# B&R Automation Studio project 2SegDemo
Automation Studio 4.10.2.37; technology packages: mapp 5.14.1, mappCockpit 5.14.0, mappControl 5.14.1, mappMotion 5.14.2, mappView 5.14.2

## Configuration 1685

CPU X20CP1685, AutomationRuntime C4.90, Build 6.3.0, Safety 1.10, Vc V4.72.2

### Task classes (Cpu.sw)
```
Cyclic#1 (cycle 1000 us, tolerance 0 us):
  6DCtrl <- Source.6DCtrl.6DCtrl.prg
  VarDemos <- Source.Demos.VarDemos.prg
  AntiSlosh <- Source.Demos.AntiSlosh.prg
Cyclic#3:
  Main <- Source.Main.Main.prg
Cyclic#4:
  Recovery <- Source.ShuttleCtrl.Recovery.prg
Cyclic#8 (cycle 1000 us):
  Vis <- Source.Auxil.Vis.prg
  MacroLoad <- Source.6DCtrl.MacroLoad.prg
  Monitor6D <- Source.Auxil.Monitor6D.prg
DataObjects: McAcpSys
Binaries: mvLoader, McMechSys, McProfGen, TCData, McAcpSim, mCoWebSc, FWRules, McAcpDrv, udbdef, TCLang, arcoal, arflatprv, arsvcreg, OpcUaSrv, Role, arconfig, Settings, User, asfw, ashwd, Config_1, ashwac, sysconf, Config, Config_2, iomap, TC, TraceConfi, Config_3, Config_4, Hierarchy
Libraries: runtime, brsystem, sys_lib, CoTrace, FileIO, AsZip, McPureVAx, operator, astime, AsIecCon, standard, McAcp6D, AsMath, AsXml, AsBrStr, AsIODiag, LoggingLib, asstring, ArEventLog, AsTCP, snprintf, MTTypes, AsBrMath, McBase, McAcpAx, McAxis, MpAxis, MpBase, MpAudit, MpRecipe, MpFile, MTFilter, MTBasics, MpServer, MpAlarmX, SlFreeBase, MTProfile, asepl, aruser, dataobj, powerlnk, arssl, asusb, WFilter, asarlog, asmem, asarprof, asio, McPathGen, McProgInt, McAxGroup, MpRobotics, McAcpTrak
```

### Hardware
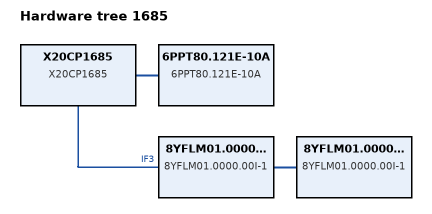
```
6PPT80.121E-10A : 6PPT80.121E-10A v1.0.2.0  [ETH1 -> X20CP1685.IF2 [Cable Type=PowerlinkCable, Length=10, Version=1.0.0.3]]
  Terminal = true
  Mode = Manual
  InternetAddress = 192.168.10.85
  Subnetmask = 255.255.255.0
  PasswordVNC = 
  PasswordCIFS = 
  PasswordService = 
8YFLM01.0000.00I-1 : 8YFLM01.0000.00I-1 v0.0.0.1  [PLK1 -> X20CP1685.IF3 (NodeNumber=101) [Cable Type=PowerlinkCable, Length=10, Version=1.0.0.3]; PLK2 -> 8YFLM01.0000.00I-1a.PLK1 (NodeNumber=101) [Cable Type=PowerlinkCable, Length=10, Version=1.0.0.3]]
  Supervision = off
8YFLM01.0000.00I-1a : 8YFLM01.0000.00I-1 v0.0.0.1 (Disabled=true)  [PLK1 -> 8YFLM01.0000.00I-1.PLK2 (NodeNumber=102) [Cable Type=PowerlinkCable, Length=10, Version=1.0.0.3]]
  Supervision = off
X20CP1685 : X20CP1685 v1.4.0.0
  Connector IF2:
    ActivateDevice = 1
    Mode = Manual
    InternetAddress = 192.168.10.82
    SubnetMask = 255.255.255.0
    ActivateSnmp = 2
  Connector IF3:
    CycleTime = 1000
  Connector IF6:
    ActivateX2X = 0
  ConfigurationID = OnsiteDemo_1685
  UserPartitionSize = 10
  TimerDeviceType = EPLX2X
  TimerDevice = X20CP1685.IF3
  Cyclic1Duration = 1000
  Cyclic1Tolerance = 0
  Cyclic1Stack = 75536
  Cyclic1Output = 1
  Cyclic2Duration = 10000
  Cyclic2Tolerance = 10000
  Cyclic8Duration = 1000
  FileDevice1
  FileDeviceName1 = CNC_PrgDir
  FileDevicePath1 = F:/Programs
  FileDevice2
  FileDeviceName2 = 6DMacro
  FileDevicePath2 = F:/Macros
  FtpUser1
  FtpUsername1 = user
  FtpUserPassword1 = OnC+KhD/SpTljM37peNi/Txa+vmo0PgBkRCvsZXBTJk=  // user
  FtpUserSalt1 = 0mgKB/Te
  FTPAccessRight1 = 0
  ActivateOpcUa = 1
  OpcUaPort = 4841
  OpcUaInformationModels_PV_Version = 2
```

### IoMap.iom - X20CP1685/IoMap.iom
```iecst
VAR_CONFIG
	Cyclic#1.::FBin[0] AT %IW."8YFLM01.0000.00I-1".EPL_FB_IN_0_I2007_S01;
	Cyclic#1.::FBin[1] AT %IW."8YFLM01.0000.00I-1".EPL_FB_IN_1_I2007_S02;
	Cyclic#1.::FBin[10] AT %IW."8YFLM01.0000.00I-1".EPL_FB_IN_10_I2007_S0B;
	Cyclic#1.::FBin[100] AT %IW."8YFLM01.0000.00I-1".EPL_FB_IN_100_I2007_S65;
	Cyclic#1.::FBin[101] AT %IW."8YFLM01.0000.00I-1".EPL_FB_IN_101_I2007_S66;
	Cyclic#1.::FBin[102] AT %IW."8YFLM01.0000.00I-1".EPL_FB_IN_102_I2007_S67;
	Cyclic#1.::FBin[103] AT %IW."8YFLM01.0000.00I-1".EPL_FB_IN_103_I2007_S68;
	Cyclic#1.::FBin[104] AT %IW."8YFLM01.0000.00I-1".EPL_FB_IN_104_I2007_S69;
	Cyclic#1.::FBin[105] AT %IW."8YFLM01.0000.00I-1".EPL_FB_IN_105_I2007_S6A;
	Cyclic#1.::FBin[106] AT %IW."8YFLM01.0000.00I-1".EPL_FB_IN_106_I2007_S6B;
	Cyclic#1.::FBin[107] AT %IW."8YFLM01.0000.00I-1".EPL_FB_IN_107_I2007_S6C;
	Cyclic#1.::FBin[108] AT %IW."8YFLM01.0000.00I-1".EPL_FB_IN_108_I2007_S6D;
	Cyclic#1.::FBin[109] AT %IW."8YFLM01.0000.00I-1".EPL_FB_IN_109_I2007_S6E;
	Cyclic#1.::FBin[11] AT %IW."8YFLM01.0000.00I-1".EPL_FB_IN_11_I2007_S0C;
	Cyclic#1.::FBin[110] AT %IW."8YFLM01.0000.00I-1".EPL_FB_IN_110_I2007_S6F;
	Cyclic#1.::FBin[111] AT %IW."8YFLM01.0000.00I-1".EPL_FB_IN_111_I2007_S70;
	Cyclic#1.::FBin[112] AT %IW."8YFLM01.0000.00I-1".EPL_FB_IN_112_I2007_S71;
	Cyclic#1.::FBin[113] AT %IW."8YFLM01.0000.00I-1".EPL_FB_IN_113_I2007_S72;
	Cyclic#1.::FBin[114] AT %IW."8YFLM01.0000.00I-1".EPL_FB_IN_114_I2007_S73;
	Cyclic#1.::FBin[115] AT %IW."8YFLM01.0000.00I-1".EPL_FB_IN_115_I2007_S74;
	Cyclic#1.::FBin[116] AT %IW."8YFLM01.0000.00I-1".EPL_FB_IN_116_I2007_S75;
	Cyclic#1.::FBin[117] AT %IW."8YFLM01.0000.00I-1".EPL_FB_IN_117_I2007_S76;
	Cyclic#1.::FBin[118] AT %IW."8YFLM01.0000.00I-1".EPL_FB_IN_118_I2007_S77;
	Cyclic#1.::FBin[119] AT %IW."8YFLM01.0000.00I-1".EPL_FB_IN_119_I2007_S78;
	Cyclic#1.::FBin[12] AT %IW."8YFLM01.0000.00I-1".EPL_FB_IN_12_I2007_S0D;
	Cyclic#1.::FBin[120] AT %IW."8YFLM01.0000.00I-1".EPL_FB_IN_120_I2007_S79;
	Cyclic#1.::FBin[121] AT %IW."8YFLM01.0000.00I-1".EPL_FB_IN_121_I2007_S7A;
	Cyclic#1.::FBin[122] AT %IW."8YFLM01.0000.00I-1".EPL_FB_IN_122_I2007_S7B;
	Cyclic#1.::FBin[123] AT %IW."8YFLM01.0000.00I-1".EPL_FB_IN_123_I2007_S7C;
	Cyclic#1.::FBin[124] AT %IW."8YFLM01.0000.00I-1".EPL_FB_IN_124_I2007_S7D;
	Cyclic#1.::FBin[125] AT %IW."8YFLM01.0000.00I-1".EPL_FB_IN_125_I2007_S7E;
	Cyclic#1.::FBin[126] AT %IW."8YFLM01.0000.00I-1".EPL_FB_IN_126_I2007_S7F;
	Cyclic#1.::FBin[127] AT %IW."8YFLM01.0000.00I-1".EPL_FB_IN_127_I2007_S80;
	Cyclic#1.::FBin[128] AT %IW."8YFLM01.0000.00I-1".EPL_FB_IN_128_I2007_S81;
	Cyclic#1.::FBin[129] AT %IW."8YFLM01.0000.00I-1".EPL_FB_IN_129_I2007_S82;
	Cyclic#1.::FBin[13] AT %IW."8YFLM01.0000.00I-1".EPL_FB_IN_13_I2007_S0E;
	Cyclic#1.::FBin[130] AT %IW."8YFLM01.0000.00I-1".EPL_FB_IN_130_I2007_S83;
	Cyclic#1.::FBin[131] AT %IW."8YFLM01.0000.00I-1".EPL_FB_IN_131_I2007_S84;
	Cyclic#1.::FBin[132] AT %IW."8YFLM01.0000.00I-1".EPL_FB_IN_132_I2007_S85;
	Cyclic#1.::FBin[133] AT %IW."8YFLM01.0000.00I-1".EPL_FB_IN_133_I2007_S86;
	Cyclic#1.::FBin[134] AT %IW."8YFLM01.0000.00I-1".EPL_FB_IN_134_I2007_S87;
	Cyclic#1.::FBin[135] AT %IW."8YFLM01.0000.00I-1".EPL_FB_IN_135_I2007_S88;
	Cyclic#1.::FBin[136] AT %IW."8YFLM01.0000.00I-1".EPL_FB_IN_136_I2007_S89;
	Cyclic#1.::FBin[137] AT %IW."8YFLM01.0000.00I-1".EPL_FB_IN_137_I2007_S8A;
	Cyclic#1.::FBin[138] AT %IW."8YFLM01.0000.00I-1".EPL_FB_IN_138_I2007_S8B;
	Cyclic#1.::FBin[139] AT %IW."8YFLM01.0000.00I-1".EPL_FB_IN_139_I2007_S8C;
	Cyclic#1.::FBin[14] AT %IW."8YFLM01.0000.00I-1".EPL_FB_IN_14_I2007_S0F;
	Cyclic#1.::FBin[140] AT %IW."8YFLM01.0000.00I-1".EPL_FB_IN_140_I2007_S8D;
	Cyclic#1.::FBin[141] AT %IW."8YFLM01.0000.00I-1".EPL_FB_IN_141_I2007_S8E;
	Cyclic#1.::FBin[142] AT %IW."8YFLM01.0000.00I-1".EPL_FB_IN_142_I2007_S8F;
	Cyclic#1.::FBin[143] AT %IW."8YFLM01.0000.00I-1".EPL_FB_IN_143_I2007_S90;
	Cyclic#1.::FBin[144] AT %IW."8YFLM01.0000.00I-1".EPL_FB_IN_144_I2007_S91;
	Cyclic#1.::FBin[145] AT %IW."8YFLM01.0000.00I-1".EPL_FB_IN_145_I2007_S92;
	Cyclic#1.::FBin[146] AT %IW."8YFLM01.0000.00I-1".EPL_FB_IN_146_I2007_S93;
	Cyclic#1.::FBin[147] AT %IW."8YFLM01.0000.00I-1".EPL_FB_IN_147_I2007_S94;
	Cyclic#1.::FBin[148] AT %IW."8YFLM01.0000.00I-1".EPL_FB_IN_148_I2007_S95;
	Cyclic#1.::FBin[149] AT %IW."8YFLM01.0000.00I-1".EPL_FB_IN_149_I2007_S96;
	Cyclic#1.::FBin[15] AT %IW."8YFLM01.0000.00I-1".EPL_FB_IN_15_I2007_S10;
	Cyclic#1.::FBin[150] AT %IW."8YFLM01.0000.00I-1".EPL_FB_IN_150_I2007_S97;
	Cyclic#1.::FBin[151] AT %IW."8YFLM01.0000.00I-1".EPL_FB_IN_151_I2007_S98;
	Cyclic#1.::FBin[152] AT %IW."8YFLM01.0000.00I-1".EPL_FB_IN_152_I2007_S99;
	Cyclic#1.::FBin[153] AT %IW."8YFLM01.0000.00I-1".EPL_FB_IN_153_I2007_S9A;
	Cyclic#1.::FBin[154] AT %IW."8YFLM01.0000.00I-1".EPL_FB_IN_154_I2007_S9B;
	Cyclic#1.::FBin[155] AT %IW."8YFLM01.0000.00I-1".EPL_FB_IN_155_I2007_S9C;
	Cyclic#1.::FBin[156] AT %IW."8YFLM01.0000.00I-1".EPL_FB_IN_156_I2007_S9D;
	Cyclic#1.::FBin[157] AT %IW."8YFLM01.0000.00I-1".EPL_FB_IN_157_I2007_S9E;
	Cyclic#1.::FBin[158] AT %IW."8YFLM01.0000.00I-1".EPL_FB_IN_158_I2007_S9F;
	Cyclic#1.::FBin[159] AT %IW."8YFLM01.0000.00I-1".EPL_FB_IN_159_I2007_SA0;
	Cyclic#1.::FBin[16] AT %IW."8YFLM01.0000.00I-1".EPL_FB_IN_16_I2007_S11;
	Cyclic#1.::FBin[160] AT %IW."8YFLM01.0000.00I-1".EPL_FB_IN_160_I2007_SA1;
	Cyclic#1.::FBin[161] AT %IW."8YFLM01.0000.00I-1".EPL_FB_IN_161_I2007_SA2;
	Cyclic#1.::FBin[162] AT %IW."8YFLM01.0000.00I-1".EPL_FB_IN_162_I2007_SA3;
	Cyclic#1.::FBin[163] AT %IW."8YFLM01.0000.00I-1".EPL_FB_IN_163_I2007_SA4;
	Cyclic#1.::FBin[164] AT %IW."8YFLM01.0000.00I-1".EPL_FB_IN_164_I2007_SA5;
	Cyclic#1.::FBin[165] AT %IW."8YFLM01.0000.00I-1".EPL_FB_IN_165_I2007_SA6;
	Cyclic#1.::FBin[166] AT %IW."8YFLM01.0000.00I-1".EPL_FB_IN_166_I2007_SA7;
	Cyclic#1.::FBin[167] AT %IW."8YFLM01.0000.00I-1".EPL_FB_IN_167_I2007_SA8;
	Cyclic#1.::FBin[168] AT %IW."8YFLM01.0000.00I-1".EPL_FB_IN_168_I2007_SA9;
	Cyclic#1.::FBin[169] AT %IW."8YFLM01.0000.00I-1".EPL_FB_IN_169_I2007_SAA;
	Cyclic#1.::FBin[17] AT %IW."8YFLM01.0000.00I-1".EPL_FB_IN_17_I2007_S12;
	Cyclic#1.::FBin[170] AT %IW."8YFLM01.0000.00I-1".EPL_FB_IN_170_I2007_SAB;
	Cyclic#1.::FBin[171] AT %IW."8YFLM01.0000.00I-1".EPL_FB_IN_171_I2007_SAC;
	Cyclic#1.::FBin[172] AT %IW."8YFLM01.0000.00I-1".EPL_FB_IN_172_I2007_SAD;
	Cyclic#1.::FBin[173] AT %IW."8YFLM01.0000.00I-1".EPL_FB_IN_173_I2007_SAE;
	Cyclic#1.::FBin[174] AT %IW."8YFLM01.0000.00I-1".EPL_FB_IN_174_I2007_SAF;
	Cyclic#1.::FBin[175] AT %IW."8YFLM01.0000.00I-1".EPL_FB_IN_175_I2007_SB0;
	Cyclic#1.::FBin[176] AT %IW."8YFLM01.0000.00I-1".EPL_FB_IN_176_I2007_SB1;
	Cyclic#1.::FBin[177] AT %IW."8YFLM01.0000.00I-1".EPL_FB_IN_177_I2007_SB2;
	Cyclic#1.::FBin[178] AT %IW."8YFLM01.0000.00I-1".EPL_FB_IN_178_I2007_SB3;
	Cyclic#1.::FBin[179] AT %IW."8YFLM01.0000.00I-1".EPL_FB_IN_179_I2007_SB4;
	Cyclic#1.::FBin[18] AT %IW."8YFLM01.0000.00I-1".EPL_FB_IN_18_I2007_S13;
	Cyclic#1.::FBin[180] AT %IW."8YFLM01.0000.00I-1".EPL_FB_IN_180_I2007_SB5;
	Cyclic#1.::FBin[181] AT %IW."8YFLM01.0000.00I-1".EPL_FB_IN_181_I2007_SB6;
	Cyclic#1.::FBin[182] AT %IW."8YFLM01.0000.00I-1".EPL_FB_IN_182_I2007_SB7;
	Cyclic#1.::FBin[183] AT %IW."8YFLM01.0000.00I-1".EPL_FB_IN_183_I2007_SB8;
	Cyclic#1.::FBin[184] AT %IW."8YFLM01.0000.00I-1".EPL_FB_IN_184_I2007_SB9;
	Cyclic#1.::FBin[185] AT %IW."8YFLM01.0000.00I-1".EPL_FB_IN_185_I2007_SBA;
	Cyclic#1.::FBin[186] AT %IW."8YFLM01.0000.00I-1".EPL_FB_IN_186_I2007_SBB;
	Cyclic#1.::FBin[187] AT %IW."8YFLM01.0000.00I-1".EPL_FB_IN_187_I2007_SBC;
	Cyclic#1.::FBin[188] AT %IW."8YFLM01.0000.00I-1".EPL_FB_IN_188_I2007_SBD;
	Cyclic#1.::FBin[189] AT %IW."8YFLM01.0000.00I-1".EPL_FB_IN_189_I2007_SBE;
	Cyclic#1.::FBin[19] AT %IW."8YFLM01.0000.00I-1".EPL_FB_IN_19_I2007_S14;
	Cyclic#1.::FBin[190] AT %IW."8YFLM01.0000.00I-1".EPL_FB_IN_190_I2007_SBF;
	Cyclic#1.::FBin[191] AT %IW."8YFLM01.0000.00I-1".EPL_FB_IN_191_I2007_SC0;
	Cyclic#1.::FBin[192] AT %IW."8YFLM01.0000.00I-1".EPL_FB_IN_192_I2007_SC1;
	Cyclic#1.::FBin[193] AT %IW."8YFLM01.0000.00I-1".EPL_FB_IN_193_I2007_SC2;
	Cyclic#1.::FBin[194] AT %IW."8YFLM01.0000.00I-1".EPL_FB_IN_194_I2007_SC3;
	Cyclic#1.::FBin[195] AT %IW."8YFLM01.0000.00I-1".EPL_FB_IN_195_I2007_SC4;
	Cyclic#1.::FBin[196] AT %IW."8YFLM01.0000.00I-1".EPL_FB_IN_196_I2007_SC5;
	Cyclic#1.::FBin[197] AT %IW."8YFLM01.0000.00I-1".EPL_FB_IN_197_I2007_SC6;
	Cyclic#1.::FBin[198] AT %IW."8YFLM01.0000.00I-1".EPL_FB_IN_198_I2007_SC7;
	Cyclic#1.::FBin[199] AT %IW."8YFLM01.0000.00I-1".EPL_FB_IN_199_I2007_SC8;
	Cyclic#1.::FBin[2] AT %IW."8YFLM01.0000.00I-1".EPL_FB_IN_2_I2007_S03;
	Cyclic#1.::FBin[20] AT %IW."8YFLM01.0000.00I-1".EPL_FB_IN_20_I2007_S15;
	Cyclic#1.::FBin[21] AT %IW."8YFLM01.0000.00I-1".EPL_FB_IN_21_I2007_S16;
	Cyclic#1.::FBin[22] AT %IW."8YFLM01.0000.00I-1".EPL_FB_IN_22_I2007_S17;
	Cyclic#1.::FBin[23] AT %IW."8YFLM01.0000.00I-1".EPL_FB_IN_23_I2007_S18;
	Cyclic#1.::FBin[24] AT %IW."8YFLM01.0000.00I-1".EPL_FB_IN_24_I2007_S19;
	Cyclic#1.::FBin[25] AT %IW."8YFLM01.0000.00I-1".EPL_FB_IN_25_I2007_S1A;
	Cyclic#1.::FBin[26] AT %IW."8YFLM01.0000.00I-1".EPL_FB_IN_26_I2007_S1B;
	Cyclic#1.::FBin[27] AT %IW."8YFLM01.0000.00I-1".EPL_FB_IN_27_I2007_S1C;
	Cyclic#1.::FBin[28] AT %IW."8YFLM01.0000.00I-1".EPL_FB_IN_28_I2007_S1D;
	Cyclic#1.::FBin[29] AT %IW."8YFLM01.0000.00I-1".EPL_FB_IN_29_I2007_S1E;
	Cyclic#1.::FBin[3] AT %IW."8YFLM01.0000.00I-1".EPL_FB_IN_3_I2007_S04;
	Cyclic#1.::FBin[30] AT %IW."8YFLM01.0000.00I-1".EPL_FB_IN_30_I2007_S1F;
	Cyclic#1.::FBin[31] AT %IW."8YFLM01.0000.00I-1".EPL_FB_IN_31_I2007_S20;
	Cyclic#1.::FBin[32] AT %IW."8YFLM01.0000.00I-1".EPL_FB_IN_32_I2007_S21;
	Cyclic#1.::FBin[33] AT %IW."8YFLM01.0000.00I-1".EPL_FB_IN_33_I2007_S22;
	Cyclic#1.::FBin[34] AT %IW."8YFLM01.0000.00I-1".EPL_FB_IN_34_I2007_S23;
	Cyclic#1.::FBin[35] AT %IW."8YFLM01.0000.00I-1".EPL_FB_IN_35_I2007_S24;
	Cyclic#1.::FBin[36] AT %IW."8YFLM01.0000.00I-1".EPL_FB_IN_36_I2007_S25;
	Cyclic#1.::FBin[37] AT %IW."8YFLM01.0000.00I-1".EPL_FB_IN_37_I2007_S26;
	Cyclic#1.::FBin[38] AT %IW."8YFLM01.0000.00I-1".EPL_FB_IN_38_I2007_S27;
	Cyclic#1.::FBin[39] AT %IW."8YFLM01.0000.00I-1".EPL_FB_IN_39_I2007_S28;
	Cyclic#1.::FBin[4] AT %IW."8YFLM01.0000.00I-1".EPL_FB_IN_4_I2007_S05;
	Cyclic#1.::FBin[40] AT %IW."8YFLM01.0000.00I-1".EPL_FB_IN_40_I2007_S29;
	Cyclic#1.::FBin[41] AT %IW."8YFLM01.0000.00I-1".EPL_FB_IN_41_I2007_S2A;
	Cyclic#1.::FBin[42] AT %IW."8YFLM01.0000.00I-1".EPL_FB_IN_42_I2007_S2B;
	Cyclic#1.::FBin[43] AT %IW."8YFLM01.0000.00I-1".EPL_FB_IN_43_I2007_S2C;
	Cyclic#1.::FBin[44] AT %IW."8YFLM01.0000.00I-1".EPL_FB_IN_44_I2007_S2D;
	Cyclic#1.::FBin[45] AT %IW."8YFLM01.0000.00I-1".EPL_FB_IN_45_I2007_S2E;
	Cyclic#1.::FBin[46] AT %IW."8YFLM01.0000.00I-1".EPL_FB_IN_46_I2007_S2F;
	Cyclic#1.::FBin[47] AT %IW."8YFLM01.0000.00I-1".EPL_FB_IN_47_I2007_S30;
	Cyclic#1.::FBin[48] AT %IW."8YFLM01.0000.00I-1".EPL_FB_IN_48_I2007_S31;
	Cyclic#1.::FBin[49] AT %IW."8YFLM01.0000.00I-1".EPL_FB_IN_49_I2007_S32;
	Cyclic#1.::FBin[5] AT %IW."8YFLM01.0000.00I-1".EPL_FB_IN_5_I2007_S06;
	Cyclic#1.::FBin[50] AT %IW."8YFLM01.0000.00I-1".EPL_FB_IN_50_I2007_S33;
	Cyclic#1.::FBin[51] AT %IW."8YFLM01.0000.00I-1".EPL_FB_IN_51_I2007_S34;
	Cyclic#1.::FBin[52] AT %IW."8YFLM01.0000.00I-1".EPL_FB_IN_52_I2007_S35;
	Cyclic#1.::FBin[53] AT %IW."8YFLM01.0000.00I-1".EPL_FB_IN_53_I2007_S36;
	Cyclic#1.::FBin[54] AT %IW."8YFLM01.0000.00I-1".EPL_FB_IN_54_I2007_S37;
	Cyclic#1.::FBin[55] AT %IW."8YFLM01.0000.00I-1".EPL_FB_IN_55_I2007_S38;
	Cyclic#1.::FBin[56] AT %IW."8YFLM01.0000.00I-1".EPL_FB_IN_56_I2007_S39;
	Cyclic#1.::FBin[57] AT %IW."8YFLM01.0000.00I-1".EPL_FB_IN_57_I2007_S3A;
	Cyclic#1.::FBin[58] AT %IW."8YFLM01.0000.00I-1".EPL_FB_IN_58_I2007_S3B;
	Cyclic#1.::FBin[59] AT %IW."8YFLM01.0000.00I-1".EPL_FB_IN_59_I2007_S3C;
	Cyclic#1.::FBin[6] AT %IW."8YFLM01.0000.00I-1".EPL_FB_IN_6_I2007_S07;
	Cyclic#1.::FBin[60] AT %IW."8YFLM01.0000.00I-1".EPL_FB_IN_60_I2007_S3D;
	Cyclic#1.::FBin[61] AT %IW."8YFLM01.0000.00I-1".EPL_FB_IN_61_I2007_S3E;
	Cyclic#1.::FBin[62] AT %IW."8YFLM01.0000.00I-1".EPL_FB_IN_62_I2007_S3F;
	Cyclic#1.::FBin[63] AT %IW."8YFLM01.0000.00I-1".EPL_FB_IN_63_I2007_S40;
	Cyclic#1.::FBin[64] AT %IW."8YFLM01.0000.00I-1".EPL_FB_IN_64_I2007_S41;
	Cyclic#1.::FBin[65] AT %IW."8YFLM01.0000.00I-1".EPL_FB_IN_65_I2007_S42;
	Cyclic#1.::FBin[66] AT %IW."8YFLM01.0000.00I-1".EPL_FB_IN_66_I2007_S43;
	Cyclic#1.::FBin[67] AT %IW."8YFLM01.0000.00I-1".EPL_FB_IN_67_I2007_S44;
	Cyclic#1.::FBin[68] AT %IW."8YFLM01.0000.00I-1".EPL_FB_IN_68_I2007_S45;
	Cyclic#1.::FBin[69] AT %IW."8YFLM01.0000.00I-1".EPL_FB_IN_69_I2007_S46;
	Cyclic#1.::FBin[7] AT %IW."8YFLM01.0000.00I-1".EPL_FB_IN_7_I2007_S08;
	Cyclic#1.::FBin[70] AT %IW."8YFLM01.0000.00I-1".EPL_FB_IN_70_I2007_S47;
	Cyclic#1.::FBin[71] AT %IW."8YFLM01.0000.00I-1".EPL_FB_IN_71_I2007_S48;
	Cyclic#1.::FBin[72] AT %IW."8YFLM01.0000.00I-1".EPL_FB_IN_72_I2007_S49;
	Cyclic#1.::FBin[73] AT %IW."8YFLM01.0000.00I-1".EPL_FB_IN_73_I2007_S4A;
	Cyclic#1.::FBin[74] AT %IW."8YFLM01.0000.00I-1".EPL_FB_IN_74_I2007_S4B;
	Cyclic#1.::FBin[75] AT %IW."8YFLM01.0000.00I-1".EPL_FB_IN_75_I2007_S4C;
	Cyclic#1.::FBin[76] AT %IW."8YFLM01.0000.00I-1".EPL_FB_IN_76_I2007_S4D;
	Cyclic#1.::FBin[77] AT %IW."8YFLM01.0000.00I-1".EPL_FB_IN_77_I2007_S4E;
	Cyclic#1.::FBin[78] AT %IW."8YFLM01.0000.00I-1".EPL_FB_IN_78_I2007_S4F;
	Cyclic#1.::FBin[79] AT %IW."8YFLM01.0000.00I-1".EPL_FB_IN_79_I2007_S50;
	Cyclic#1.::FBin[8] AT %IW."8YFLM01.0000.00I-1".EPL_FB_IN_8_I2007_S09;
	Cyclic#1.::FBin[80] AT %IW."8YFLM01.0000.00I-1".EPL_FB_IN_80_I2007_S51;
	Cyclic#1.::FBin[81] AT %IW."8YFLM01.0000.00I-1".EPL_FB_IN_81_I2007_S52;
	Cyclic#1.::FBin[82] AT %IW."8YFLM01.0000.00I-1".EPL_FB_IN_82_I2007_S53;
	Cyclic#1.::FBin[83] AT %IW."8YFLM01.0000.00I-1".EPL_FB_IN_83_I2007_S54;
	Cyclic#1.::FBin[84] AT %IW."8YFLM01.0000.00I-1".EPL_FB_IN_84_I2007_S55;
	Cyclic#1.::FBin[85] AT %IW."8YFLM01.0000.00I-1".EPL_FB_IN_85_I2007_S56;
	Cyclic#1.::FBin[86] AT %IW."8YFLM01.0000.00I-1".EPL_FB_IN_86_I2007_S57;
	Cyclic#1.::FBin[87] AT %IW."8YFLM01.0000.00I-1".EPL_FB_IN_87_I2007_S58;
	Cyclic#1.::FBin[88] AT %IW."8YFLM01.0000.00I-1".EPL_FB_IN_88_I2007_S59;
	Cyclic#1.::FBin[89] AT %IW."8YFLM01.0000.00I-1".EPL_FB_IN_89_I2007_S5A;
	Cyclic#1.::FBin[9] AT %IW."8YFLM01.0000.00I-1".EPL_FB_IN_9_I2007_S0A;
	Cyclic#1.::FBin[90] AT %IW."8YFLM01.0000.00I-1".EPL_FB_IN_90_I2007_S5B;
	Cyclic#1.::FBin[91] AT %IW."8YFLM01.0000.00I-1".EPL_FB_IN_91_I2007_S5C;
	Cyclic#1.::FBin[92] AT %IW."8YFLM01.0000.00I-1".EPL_FB_IN_92_I2007_S5D;
	Cyclic#1.::FBin[93] AT %IW."8YFLM01.0000.00I-1".EPL_FB_IN_93_I2007_S5E;
	Cyclic#1.::FBin[94] AT %IW."8YFLM01.0000.00I-1".EPL_FB_IN_94_I2007_S5F;
	Cyclic#1.::FBin[95] AT %IW."8YFLM01.0000.00I-1".EPL_FB_IN_95_I2007_S60;
	Cyclic#1.::FBin[96] AT %IW."8YFLM01.0000.00I-1".EPL_FB_IN_96_I2007_S61;
	Cyclic#1.::FBin[97] AT %IW."8YFLM01.0000.00I-1".EPL_FB_IN_97_I2007_S62;
	Cyclic#1.::FBin[98] AT %IW."8YFLM01.0000.00I-1".EPL_FB_IN_98_I2007_S63;
	Cyclic#1.::FBin[99] AT %IW."8YFLM01.0000.00I-1".EPL_FB_IN_99_I2007_S64;
	Cyclic#1.::FBout[0] AT %QW."8YFLM01.0000.00I-1".EPL_FB_OUT_0_I2008_S01Out;
	Cyclic#1.::FBout[1] AT %QW."8YFLM01.0000.00I-1".EPL_FB_OUT_1_I2008_S02Out;
	Cyclic#1.::FBout[10] AT %QW."8YFLM01.0000.00I-1".EPL_FB_OUT_10_I2008_S0BOut;
	Cyclic#1.::FBout[100] AT %QW."8YFLM01.0000.00I-1".EPL_FB_OUT_100_I2008_S65Out;
	Cyclic#1.::FBout[101] AT %QW."8YFLM01.0000.00I-1".EPL_FB_OUT_101_I2008_S66Out;
	Cyclic#1.::FBout[102] AT %QW."8YFLM01.0000.00I-1".EPL_FB_OUT_102_I2008_S67Out;
	Cyclic#1.::FBout[103] AT %QW."8YFLM01.0000.00I-1".EPL_FB_OUT_103_I2008_S68Out;
	Cyclic#1.::FBout[104] AT %QW."8YFLM01.0000.00I-1".EPL_FB_OUT_104_I2008_S69Out;
	Cyclic#1.::FBout[105] AT %QW."8YFLM01.0000.00I-1".EPL_FB_OUT_105_I2008_S6AOut;
	Cyclic#1.::FBout[106] AT %QW."8YFLM01.0000.00I-1".EPL_FB_OUT_106_I2008_S6BOut;
	Cyclic#1.::FBout[107] AT %QW."8YFLM01.0000.00I-1".EPL_FB_OUT_107_I2008_S6COut;
	Cyclic#1.::FBout[108] AT %QW."8YFLM01.0000.00I-1".EPL_FB_OUT_108_I2008_S6DOut;
	Cyclic#1.::FBout[109] AT %QW."8YFLM01.0000.00I-1".EPL_FB_OUT_109_I2008_S6EOut;
	Cyclic#1.::FBout[11] AT %QW."8YFLM01.0000.00I-1".EPL_FB_OUT_11_I2008_S0COut;
	Cyclic#1.::FBout[110] AT %QW."8YFLM01.0000.00I-1".EPL_FB_OUT_110_I2008_S6FOut;
	Cyclic#1.::FBout[111] AT %QW."8YFLM01.0000.00I-1".EPL_FB_OUT_111_I2008_S70Out;
	Cyclic#1.::FBout[112] AT %QW."8YFLM01.0000.00I-1".EPL_FB_OUT_112_I2008_S71Out;
	Cyclic#1.::FBout[113] AT %QW."8YFLM01.0000.00I-1".EPL_FB_OUT_113_I2008_S72Out;
	Cyclic#1.::FBout[114] AT %QW."8YFLM01.0000.00I-1".EPL_FB_OUT_114_I2008_S73Out;
	Cyclic#1.::FBout[115] AT %QW."8YFLM01.0000.00I-1".EPL_FB_OUT_115_I2008_S74Out;
	Cyclic#1.::FBout[116] AT %QW."8YFLM01.0000.00I-1".EPL_FB_OUT_116_I2008_S75Out;
	Cyclic#1.::FBout[117] AT %QW."8YFLM01.0000.00I-1".EPL_FB_OUT_117_I2008_S76Out;
	Cyclic#1.::FBout[118] AT %QW."8YFLM01.0000.00I-1".EPL_FB_OUT_118_I2008_S77Out;
	Cyclic#1.::FBout[119] AT %QW."8YFLM01.0000.00I-1".EPL_FB_OUT_119_I2008_S78Out;
	Cyclic#1.::FBout[12] AT %QW."8YFLM01.0000.00I-1".EPL_FB_OUT_12_I2008_S0DOut;
	Cyclic#1.::FBout[120] AT %QW."8YFLM01.0000.00I-1".EPL_FB_OUT_120_I2008_S79Out;
	Cyclic#1.::FBout[121] AT %QW."8YFLM01.0000.00I-1".EPL_FB_OUT_121_I2008_S7AOut;
	Cyclic#1.::FBout[122] AT %QW."8YFLM01.0000.00I-1".EPL_FB_OUT_122_I2008_S7BOut;
	Cyclic#1.::FBout[123] AT %QW."8YFLM01.0000.00I-1".EPL_FB_OUT_123_I2008_S7COut;
	Cyclic#1.::FBout[124] AT %QW."8YFLM01.0000.00I-1".EPL_FB_OUT_124_I2008_S7DOut;
	Cyclic#1.::FBout[125] AT %QW."8YFLM01.0000.00I-1".EPL_FB_OUT_125_I2008_S7EOut;
	Cyclic#1.::FBout[126] AT %QW."8YFLM01.0000.00I-1".EPL_FB_OUT_126_I2008_S7FOut;
	Cyclic#1.::FBout[127] AT %QW."8YFLM01.0000.00I-1".EPL_FB_OUT_127_I2008_S80Out;
	Cyclic#1.::FBout[128] AT %QW."8YFLM01.0000.00I-1".EPL_FB_OUT_128_I2008_S81Out;
	Cyclic#1.::FBout[129] AT %QW."8YFLM01.0000.00I-1".EPL_FB_OUT_129_I2008_S82Out;
	Cyclic#1.::FBout[13] AT %QW."8YFLM01.0000.00I-1".EPL_FB_OUT_13_I2008_S0EOut;
	Cyclic#1.::FBout[130] AT %QW."8YFLM01.0000.00I-1".EPL_FB_OUT_130_I2008_S83Out;
	Cyclic#1.::FBout[131] AT %QW."8YFLM01.0000.00I-1".EPL_FB_OUT_131_I2008_S84Out;
	Cyclic#1.::FBout[132] AT %QW."8YFLM01.0000.00I-1".EPL_FB_OUT_132_I2008_S85Out;
	Cyclic#1.::FBout[133] AT %QW."8YFLM01.0000.00I-1".EPL_FB_OUT_133_I2008_S86Out;
	Cyclic#1.::FBout[134] AT %QW."8YFLM01.0000.00I-1".EPL_FB_OUT_134_I2008_S87Out;
	Cyclic#1.::FBout[135] AT %QW."8YFLM01.0000.00I-1".EPL_FB_OUT_135_I2008_S88Out;
	Cyclic#1.::FBout[136] AT %QW."8YFLM01.0000.00I-1".EPL_FB_OUT_136_I2008_S89Out;
	Cyclic#1.::FBout[137] AT %QW."8YFLM01.0000.00I-1".EPL_FB_OUT_137_I2008_S8AOut;
	Cyclic#1.::FBout[138] AT %QW."8YFLM01.0000.00I-1".EPL_FB_OUT_138_I2008_S8BOut;
	Cyclic#1.::FBout[139] AT %QW."8YFLM01.0000.00I-1".EPL_FB_OUT_139_I2008_S8COut;
	Cyclic#1.::FBout[14] AT %QW."8YFLM01.0000.00I-1".EPL_FB_OUT_14_I2008_S0FOut;
	Cyclic#1.::FBout[140] AT %QW."8YFLM01.0000.00I-1".EPL_FB_OUT_140_I2008_S8DOut;
	Cyclic#1.::FBout[141] AT %QW."8YFLM01.0000.00I-1".EPL_FB_OUT_141_I2008_S8EOut;
	Cyclic#1.::FBout[142] AT %QW."8YFLM01.0000.00I-1".EPL_FB_OUT_142_I2008_S8FOut;
	Cyclic#1.::FBout[143] AT %QW."8YFLM01.0000.00I-1".EPL_FB_OUT_143_I2008_S90Out;
	Cyclic#1.::FBout[144] AT %QW."8YFLM01.0000.00I-1".EPL_FB_OUT_144_I2008_S91Out;
	Cyclic#1.::FBout[145] AT %QW."8YFLM01.0000.00I-1".EPL_FB_OUT_145_I2008_S92Out;
	Cyclic#1.::FBout[146] AT %QW."8YFLM01.0000.00I-1".EPL_FB_OUT_146_I2008_S93Out;
	Cyclic#1.::FBout[147] AT %QW."8YFLM01.0000.00I-1".EPL_FB_OUT_147_I2008_S94Out;
	Cyclic#1.::FBout[148] AT %QW."8YFLM01.0000.00I-1".EPL_FB_OUT_148_I2008_S95Out;
	Cyclic#1.::FBout[149] AT %QW."8YFLM01.0000.00I-1".EPL_FB_OUT_149_I2008_S96Out;
	Cyclic#1.::FBout[15] AT %QW."8YFLM01.0000.00I-1".EPL_FB_OUT_15_I2008_S10Out;
	Cyclic#1.::FBout[150] AT %QW."8YFLM01.0000.00I-1".EPL_FB_OUT_150_I2008_S97Out;
	Cyclic#1.::FBout[151] AT %QW."8YFLM01.0000.00I-1".EPL_FB_OUT_151_I2008_S98Out;
	Cyclic#1.::FBout[152] AT %QW."8YFLM01.0000.00I-1".EPL_FB_OUT_152_I2008_S99Out;
	Cyclic#1.::FBout[153] AT %QW."8YFLM01.0000.00I-1".EPL_FB_OUT_153_I2008_S9AOut;
	Cyclic#1.::FBout[154] AT %QW."8YFLM01.0000.00I-1".EPL_FB_OUT_154_I2008_S9BOut;
	Cyclic#1.::FBout[155] AT %QW."8YFLM01.0000.00I-1".EPL_FB_OUT_155_I2008_S9COut;
	Cyclic#1.::FBout[156] AT %QW."8YFLM01.0000.00I-1".EPL_FB_OUT_156_I2008_S9DOut;
	Cyclic#1.::FBout[157] AT %QW."8YFLM01.0000.00I-1".EPL_FB_OUT_157_I2008_S9EOut;
	Cyclic#1.::FBout[158] AT %QW."8YFLM01.0000.00I-1".EPL_FB_OUT_158_I2008_S9FOut;
	Cyclic#1.::FBout[159] AT %QW."8YFLM01.0000.00I-1".EPL_FB_OUT_159_I2008_SA0Out;
	Cyclic#1.::FBout[16] AT %QW."8YFLM01.0000.00I-1".EPL_FB_OUT_16_I2008_S11Out;
	Cyclic#1.::FBout[160] AT %QW."8YFLM01.0000.00I-1".EPL_FB_OUT_160_I2008_SA1Out;
	Cyclic#1.::FBout[161] AT %QW."8YFLM01.0000.00I-1".EPL_FB_OUT_161_I2008_SA2Out;
	Cyclic#1.::FBout[162] AT %QW."8YFLM01.0000.00I-1".EPL_FB_OUT_162_I2008_SA3Out;
	Cyclic#1.::FBout[163] AT %QW."8YFLM01.0000.00I-1".EPL_FB_OUT_163_I2008_SA4Out;
	Cyclic#1.::FBout[164] AT %QW."8YFLM01.0000.00I-1".EPL_FB_OUT_164_I2008_SA5Out;
	Cyclic#1.::FBout[165] AT %QW."8YFLM01.0000.00I-1".EPL_FB_OUT_165_I2008_SA6Out;
	Cyclic#1.::FBout[166] AT %QW."8YFLM01.0000.00I-1".EPL_FB_OUT_166_I2008_SA7Out;
	Cyclic#1.::FBout[167] AT %QW."8YFLM01.0000.00I-1".EPL_FB_OUT_167_I2008_SA8Out;
	Cyclic#1.::FBout[168] AT %QW."8YFLM01.0000.00I-1".EPL_FB_OUT_168_I2008_SA9Out;
	Cyclic#1.::FBout[169] AT %QW."8YFLM01.0000.00I-1".EPL_FB_OUT_169_I2008_SAAOut;
	Cyclic#1.::FBout[17] AT %QW."8YFLM01.0000.00I-1".EPL_FB_OUT_17_I2008_S12Out;
	Cyclic#1.::FBout[170] AT %QW."8YFLM01.0000.00I-1".EPL_FB_OUT_170_I2008_SABOut;
	Cyclic#1.::FBout[171] AT %QW."8YFLM01.0000.00I-1".EPL_FB_OUT_171_I2008_SACOut;
	Cyclic#1.::FBout[172] AT %QW."8YFLM01.0000.00I-1".EPL_FB_OUT_172_I2008_SADOut;
	Cyclic#1.::FBout[173] AT %QW."8YFLM01.0000.00I-1".EPL_FB_OUT_173_I2008_SAEOut;
	Cyclic#1.::FBout[174] AT %QW."8YFLM01.0000.00I-1".EPL_FB_OUT_174_I2008_SAFOut;
	Cyclic#1.::FBout[175] AT %QW."8YFLM01.0000.00I-1".EPL_FB_OUT_175_I2008_SB0Out;
	Cyclic#1.::FBout[176] AT %QW."8YFLM01.0000.00I-1".EPL_FB_OUT_176_I2008_SB1Out;
	Cyclic#1.::FBout[177] AT %QW."8YFLM01.0000.00I-1".EPL_FB_OUT_177_I2008_SB2Out;
	Cyclic#1.::FBout[178] AT %QW."8YFLM01.0000.00I-1".EPL_FB_OUT_178_I2008_SB3Out;
	Cyclic#1.::FBout[179] AT %QW."8YFLM01.0000.00I-1".EPL_FB_OUT_179_I2008_SB4Out;
	Cyclic#1.::FBout[18] AT %QW."8YFLM01.0000.00I-1".EPL_FB_OUT_18_I2008_S13Out;
	Cyclic#1.::FBout[180] AT %QW."8YFLM01.0000.00I-1".EPL_FB_OUT_180_I2008_SB5Out;
	Cyclic#1.::FBout[181] AT %QW."8YFLM01.0000.00I-1".EPL_FB_OUT_181_I2008_SB6Out;
	Cyclic#1.::FBout[182] AT %QW."8YFLM01.0000.00I-1".EPL_FB_OUT_182_I2008_SB7Out;
	Cyclic#1.::FBout[183] AT %QW."8YFLM01.0000.00I-1".EPL_FB_OUT_183_I2008_SB8Out;
	Cyclic#1.::FBout[184] AT %QW."8YFLM01.0000.00I-1".EPL_FB_OUT_184_I2008_SB9Out;
	Cyclic#1.::FBout[185] AT %QW."8YFLM01.0000.00I-1".EPL_FB_OUT_185_I2008_SBAOut;
	Cyclic#1.::FBout[186] AT %QW."8YFLM01.0000.00I-1".EPL_FB_OUT_186_I2008_SBBOut;
	Cyclic#1.::FBout[187] AT %QW."8YFLM01.0000.00I-1".EPL_FB_OUT_187_I2008_SBCOut;
	Cyclic#1.::FBout[188] AT %QW."8YFLM01.0000.00I-1".EPL_FB_OUT_188_I2008_SBDOut;
	Cyclic#1.::FBout[189] AT %QW."8YFLM01.0000.00I-1".EPL_FB_OUT_189_I2008_SBEOut;
	Cyclic#1.::FBout[19] AT %QW."8YFLM01.0000.00I-1".EPL_FB_OUT_19_I2008_S14Out;
	Cyclic#1.::FBout[190] AT %QW."8YFLM01.0000.00I-1".EPL_FB_OUT_190_I2008_SBFOut;
	Cyclic#1.::FBout[191] AT %QW."8YFLM01.0000.00I-1".EPL_FB_OUT_191_I2008_SC0Out;
	Cyclic#1.::FBout[192] AT %QW."8YFLM01.0000.00I-1".EPL_FB_OUT_192_I2008_SC1Out;
	Cyclic#1.::FBout[193] AT %QW."8YFLM01.0000.00I-1".EPL_FB_OUT_193_I2008_SC2Out;
	Cyclic#1.::FBout[194] AT %QW."8YFLM01.0000.00I-1".EPL_FB_OUT_194_I2008_SC3Out;
	Cyclic#1.::FBout[195] AT %QW."8YFLM01.0000.00I-1".EPL_FB_OUT_195_I2008_SC4Out;
	Cyclic#1.::FBout[196] AT %QW."8YFLM01.0000.00I-1".EPL_FB_OUT_196_I2008_SC5Out;
	Cyclic#1.::FBout[197] AT %QW."8YFLM01.0000.00I-1".EPL_FB_OUT_197_I2008_SC6Out;
	Cyclic#1.::FBout[198] AT %QW."8YFLM01.0000.00I-1".EPL_FB_OUT_198_I2008_SC7Out;
	Cyclic#1.::FBout[199] AT %QW."8YFLM01.0000.00I-1".EPL_FB_OUT_199_I2008_SC8Out;
	Cyclic#1.::FBout[2] AT %QW."8YFLM01.0000.00I-1".EPL_FB_OUT_2_I2008_S03Out;
	Cyclic#1.::FBout[20] AT %QW."8YFLM01.0000.00I-1".EPL_FB_OUT_20_I2008_S15Out;
	Cyclic#1.::FBout[21] AT %QW."8YFLM01.0000.00I-1".EPL_FB_OUT_21_I2008_S16Out;
	Cyclic#1.::FBout[22] AT %QW."8YFLM01.0000.00I-1".EPL_FB_OUT_22_I2008_S17Out;
	Cyclic#1.::FBout[23] AT %QW."8YFLM01.0000.00I-1".EPL_FB_OUT_23_I2008_S18Out;
	Cyclic#1.::FBout[24] AT %QW."8YFLM01.0000.00I-1".EPL_FB_OUT_24_I2008_S19Out;
	Cyclic#1.::FBout[25] AT %QW."8YFLM01.0000.00I-1".EPL_FB_OUT_25_I2008_S1AOut;
	Cyclic#1.::FBout[26] AT %QW."8YFLM01.0000.00I-1".EPL_FB_OUT_26_I2008_S1BOut;
	Cyclic#1.::FBout[27] AT %QW."8YFLM01.0000.00I-1".EPL_FB_OUT_27_I2008_S1COut;
	Cyclic#1.::FBout[28] AT %QW."8YFLM01.0000.00I-1".EPL_FB_OUT_28_I2008_S1DOut;
	Cyclic#1.::FBout[29] AT %QW."8YFLM01.0000.00I-1".EPL_FB_OUT_29_I2008_S1EOut;
	Cyclic#1.::FBout[3] AT %QW."8YFLM01.0000.00I-1".EPL_FB_OUT_3_I2008_S04Out;
	Cyclic#1.::FBout[30] AT %QW."8YFLM01.0000.00I-1".EPL_FB_OUT_30_I2008_S1FOut;
	Cyclic#1.::FBout[31] AT %QW."8YFLM01.0000.00I-1".EPL_FB_OUT_31_I2008_S20Out;
	Cyclic#1.::FBout[32] AT %QW."8YFLM01.0000.00I-1".EPL_FB_OUT_32_I2008_S21Out;
	Cyclic#1.::FBout[33] AT %QW."8YFLM01.0000.00I-1".EPL_FB_OUT_33_I2008_S22Out;
	Cyclic#1.::FBout[34] AT %QW."8YFLM01.0000.00I-1".EPL_FB_OUT_34_I2008_S23Out;
	Cyclic#1.::FBout[35] AT %QW."8YFLM01.0000.00I-1".EPL_FB_OUT_35_I2008_S24Out;
	Cyclic#1.::FBout[36] AT %QW."8YFLM01.0000.00I-1".EPL_FB_OUT_36_I2008_S25Out;
	Cyclic#1.::FBout[37] AT %QW."8YFLM01.0000.00I-1".EPL_FB_OUT_37_I2008_S26Out;
	Cyclic#1.::FBout[38] AT %QW."8YFLM01.0000.00I-1".EPL_FB_OUT_38_I2008_S27Out;
	Cyclic#1.::FBout[39] AT %QW."8YFLM01.0000.00I-1".EPL_FB_OUT_39_I2008_S28Out;
	Cyclic#1.::FBout[4] AT %QW."8YFLM01.0000.00I-1".EPL_FB_OUT_4_I2008_S05Out;
	Cyclic#1.::FBout[40] AT %QW."8YFLM01.0000.00I-1".EPL_FB_OUT_40_I2008_S29Out;
	Cyclic#1.::FBout[41] AT %QW."8YFLM01.0000.00I-1".EPL_FB_OUT_41_I2008_S2AOut;
	Cyclic#1.::FBout[42] AT %QW."8YFLM01.0000.00I-1".EPL_FB_OUT_42_I2008_S2BOut;
	Cyclic#1.::FBout[43] AT %QW."8YFLM01.0000.00I-1".EPL_FB_OUT_43_I2008_S2COut;
	Cyclic#1.::FBout[44] AT %QW."8YFLM01.0000.00I-1".EPL_FB_OUT_44_I2008_S2DOut;
	Cyclic#1.::FBout[45] AT %QW."8YFLM01.0000.00I-1".EPL_FB_OUT_45_I2008_S2EOut;
	Cyclic#1.::FBout[46] AT %QW."8YFLM01.0000.00I-1".EPL_FB_OUT_46_I2008_S2FOut;
	Cyclic#1.::FBout[47] AT %QW."8YFLM01.0000.00I-1".EPL_FB_OUT_47_I2008_S30Out;
	Cyclic#1.::FBout[48] AT %QW."8YFLM01.0000.00I-1".EPL_FB_OUT_48_I2008_S31Out;
	Cyclic#1.::FBout[49] AT %QW."8YFLM01.0000.00I-1".EPL_FB_OUT_49_I2008_S32Out;
	Cyclic#1.::FBout[5] AT %QW."8YFLM01.0000.00I-1".EPL_FB_OUT_5_I2008_S06Out;
	Cyclic#1.::FBout[50] AT %QW."8YFLM01.0000.00I-1".EPL_FB_OUT_50_I2008_S33Out;
	Cyclic#1.::FBout[51] AT %QW."8YFLM01.0000.00I-1".EPL_FB_OUT_51_I2008_S34Out;
	Cyclic#1.::FBout[52] AT %QW."8YFLM01.0000.00I-1".EPL_FB_OUT_52_I2008_S35Out;
	Cyclic#1.::FBout[53] AT %QW."8YFLM01.0000.00I-1".EPL_FB_OUT_53_I2008_S36Out;
	Cyclic#1.::FBout[54] AT %QW."8YFLM01.0000.00I-1".EPL_FB_OUT_54_I2008_S37Out;
	Cyclic#1.::FBout[55] AT %QW."8YFLM01.0000.00I-1".EPL_FB_OUT_55_I2008_S38Out;
	Cyclic#1.::FBout[56] AT %QW."8YFLM01.0000.00I-1".EPL_FB_OUT_56_I2008_S39Out;
	Cyclic#1.::FBout[57] AT %QW."8YFLM01.0000.00I-1".EPL_FB_OUT_57_I2008_S3AOut;
	Cyclic#1.::FBout[58] AT %QW."8YFLM01.0000.00I-1".EPL_FB_OUT_58_I2008_S3BOut;
	Cyclic#1.::FBout[59] AT %QW."8YFLM01.0000.00I-1".EPL_FB_OUT_59_I2008_S3COut;
	Cyclic#1.::FBout[6] AT %QW."8YFLM01.0000.00I-1".EPL_FB_OUT_6_I2008_S07Out;
	Cyclic#1.::FBout[60] AT %QW."8YFLM01.0000.00I-1".EPL_FB_OUT_60_I2008_S3DOut;
	Cyclic#1.::FBout[61] AT %QW."8YFLM01.0000.00I-1".EPL_FB_OUT_61_I2008_S3EOut;
	Cyclic#1.::FBout[62] AT %QW."8YFLM01.0000.00I-1".EPL_FB_OUT_62_I2008_S3FOut;
	Cyclic#1.::FBout[63] AT %QW."8YFLM01.0000.00I-1".EPL_FB_OUT_63_I2008_S40Out;
	Cyclic#1.::FBout[64] AT %QW."8YFLM01.0000.00I-1".EPL_FB_OUT_64_I2008_S41Out;
	Cyclic#1.::FBout[65] AT %QW."8YFLM01.0000.00I-1".EPL_FB_OUT_65_I2008_S42Out;
	Cyclic#1.::FBout[66] AT %QW."8YFLM01.0000.00I-1".EPL_FB_OUT_66_I2008_S43Out;
	Cyclic#1.::FBout[67] AT %QW."8YFLM01.0000.00I-1".EPL_FB_OUT_67_I2008_S44Out;
	Cyclic#1.::FBout[68] AT %QW."8YFLM01.0000.00I-1".EPL_FB_OUT_68_I2008_S45Out;
	Cyclic#1.::FBout[69] AT %QW."8YFLM01.0000.00I-1".EPL_FB_OUT_69_I2008_S46Out;
	Cyclic#1.::FBout[7] AT %QW."8YFLM01.0000.00I-1".EPL_FB_OUT_7_I2008_S08Out;
	Cyclic#1.::FBout[70] AT %QW."8YFLM01.0000.00I-1".EPL_FB_OUT_70_I2008_S47Out;
	Cyclic#1.::FBout[71] AT %QW."8YFLM01.0000.00I-1".EPL_FB_OUT_71_I2008_S48Out;
	Cyclic#1.::FBout[72] AT %QW."8YFLM01.0000.00I-1".EPL_FB_OUT_72_I2008_S49Out;
	Cyclic#1.::FBout[73] AT %QW."8YFLM01.0000.00I-1".EPL_FB_OUT_73_I2008_S4AOut;
	Cyclic#1.::FBout[74] AT %QW."8YFLM01.0000.00I-1".EPL_FB_OUT_74_I2008_S4BOut;
	Cyclic#1.::FBout[75] AT %QW."8YFLM01.0000.00I-1".EPL_FB_OUT_75_I2008_S4COut;
	Cyclic#1.::FBout[76] AT %QW."8YFLM01.0000.00I-1".EPL_FB_OUT_76_I2008_S4DOut;
	Cyclic#1.::FBout[77] AT %QW."8YFLM01.0000.00I-1".EPL_FB_OUT_77_I2008_S4EOut;
	Cyclic#1.::FBout[78] AT %QW."8YFLM01.0000.00I-1".EPL_FB_OUT_78_I2008_S4FOut;
	Cyclic#1.::FBout[79] AT %QW."8YFLM01.0000.00I-1".EPL_FB_OUT_79_I2008_S50Out;
	Cyclic#1.::FBout[8] AT %QW."8YFLM01.0000.00I-1".EPL_FB_OUT_8_I2008_S09Out;
	Cyclic#1.::FBout[80] AT %QW."8YFLM01.0000.00I-1".EPL_FB_OUT_80_I2008_S51Out;
	Cyclic#1.::FBout[81] AT %QW."8YFLM01.0000.00I-1".EPL_FB_OUT_81_I2008_S52Out;
	Cyclic#1.::FBout[82] AT %QW."8YFLM01.0000.00I-1".EPL_FB_OUT_82_I2008_S53Out;
	Cyclic#1.::FBout[83] AT %QW."8YFLM01.0000.00I-1".EPL_FB_OUT_83_I2008_S54Out;
	Cyclic#1.::FBout[84] AT %QW."8YFLM01.0000.00I-1".EPL_FB_OUT_84_I2008_S55Out;
	Cyclic#1.::FBout[85] AT %QW."8YFLM01.0000.00I-1".EPL_FB_OUT_85_I2008_S56Out;
	Cyclic#1.::FBout[86] AT %QW."8YFLM01.0000.00I-1".EPL_FB_OUT_86_I2008_S57Out;
	Cyclic#1.::FBout[87] AT %QW."8YFLM01.0000.00I-1".EPL_FB_OUT_87_I2008_S58Out;
	Cyclic#1.::FBout[88] AT %QW."8YFLM01.0000.00I-1".EPL_FB_OUT_88_I2008_S59Out;
	Cyclic#1.::FBout[89] AT %QW."8YFLM01.0000.00I-1".EPL_FB_OUT_89_I2008_S5AOut;
	Cyclic#1.::FBout[9] AT %QW."8YFLM01.0000.00I-1".EPL_FB_OUT_9_I2008_S0AOut;
	Cyclic#1.::FBout[90] AT %QW."8YFLM01.0000.00I-1".EPL_FB_OUT_90_I2008_S5BOut;
	Cyclic#1.::FBout[91] AT %QW."8YFLM01.0000.00I-1".EPL_FB_OUT_91_I2008_S5COut;
	Cyclic#1.::FBout[92] AT %QW."8YFLM01.0000.00I-1".EPL_FB_OUT_92_I2008_S5DOut;
	Cyclic#1.::FBout[93] AT %QW."8YFLM01.0000.00I-1".EPL_FB_OUT_93_I2008_S5EOut;
	Cyclic#1.::FBout[94] AT %QW."8YFLM01.0000.00I-1".EPL_FB_OUT_94_I2008_S5FOut;
	Cyclic#1.::FBout[95] AT %QW."8YFLM01.0000.00I-1".EPL_FB_OUT_95_I2008_S60Out;
	Cyclic#1.::FBout[96] AT %QW."8YFLM01.0000.00I-1".EPL_FB_OUT_96_I2008_S61Out;
	Cyclic#1.::FBout[97] AT %QW."8YFLM01.0000.00I-1".EPL_FB_OUT_97_I2008_S62Out;
	Cyclic#1.::FBout[98] AT %QW."8YFLM01.0000.00I-1".EPL_FB_OUT_98_I2008_S63Out;
	Cyclic#1.::FBout[99] AT %QW."8YFLM01.0000.00I-1".EPL_FB_OUT_99_I2008_S64Out;

END_VAR
```

### Config_1.axis - X20CP1685/mappMotion/PureVAxis/Config_1.axis
```
Element gAxis_1 (Type=axis)
  BaseTypeIsReadOnly = 0
  BaseType = LinearBounded
    MeasurementUnit = 5066068
    MeasurementResolutionIsReadOnly = 0
    MeasurementResolution = 0.01
    CountDirectionIsReadOnly = 0
    CountDirection = Standard
  MovementLimitsIsReadOnly = 0
  MovementLimits = Internal
    Position:
      LowerLimitMin = -1.79769313486231E308
      UpperLimitMax = 1.79769313486231E308
      LowerLimit = -1000.0
      UpperLimit = 1000.0
    VelocityIsReadOnly = 0
    Velocity:
      VelocityMax = 3.4E38
      Velocity = 1000
    AccelerationIsReadOnly = 0
    Acceleration:
      AccelerationMax = 3.4E38
      Acceleration = 5000
    DecelerationIsReadOnly = 0
    Deceleration:
      DecelerationMax = 3.4E38
      Deceleration = 5000
  Alarms = None
```

### Config_2.purevaxcfg - X20CP1685/mappMotion/PureVAxis/Config_2.purevaxcfg
```
Element PureVAxCfg_1 (Type=purevaxcfg)
  TypeID = PureVAxConfig
  PureVAxis:
    AxisReference = gAxis_1
    Homing:
      Mode = Direct
        Position = 0.0
        ReferencePulse = NotUsed
      RestorePositionVariable
    JerkLimitedIsFiltered = true
    JerkFilter = Used
      MaxJerkTime = 0.1
      JerkTime = 0.1
```

## Configuration 910

CPU 5PC900.TS17-00, AutomationRuntime C4.90, Build 6.3.0, Safety 0.0, Vc V4.72.2

### Task classes (Cpu.sw)
```
Cyclic#1 (cycle 1000 us, tolerance 0 us):
  6DCtrl <- Source.6DCtrl.6DCtrl.prg
  WaveDemo <- Source.Demos.WaveDemo.prg
  AntiSlosh <- Source.Demos.AntiSlosh.prg
  VarDemos <- Source.Demos.VarDemos.prg
  ConvUnload <- (binary)
  KalmanTes1 <- (binary)
  VariedMovD <- (binary)
  MacroDemo <- (binary)
  KalmanTest <- (binary)
Cyclic#3:
  Main <- Source.Main.Main.prg
Cyclic#8 (cycle 2000 us):
  Vis <- Source.Auxil.Vis.prg
  Monitor6D <- Source.Auxil.Monitor6D.prg
  SVControl <- Source.Auxil.SVControl.prg [disabled]
  MacroLoad <- Source.6DCtrl.MacroLoad.prg
DataObjects: McAcpSys
NcDataObjects: AcpParTab
Binaries: TCLang, udbdef, FWRules, mvLoader, mCoWebSc, TCData, OpcUaSrv, arsvcreg, mcacpdrv, arflatprv, arcoal, McAcpSim, McProfGen, McMechSys, iomap, asfw, Role, ashwd, sysconf, arconfig, ashwac, User, TC, Config_1, Config_2, Config_4, Hierarchy, Config_5, Config_3, Config_6, Settings, Config, CfgRecipe, CITT_FileU, CITT_Alarm, CITT_Recip, Config_8, Config_9, Config_7, Config_10, TraceConfi
Libraries: MpAudit, MpBase, McAxGroup, McBase, McPathGen, McAxis, McProgInt, CoTrace, AsZip, FileIO, runtime, MTBasics, brsystem, MTFilter, sys_lib, MTTypes, operator, astime, AsIecCon, standard, McAcp6D, AsXml, AsBrStr, AsIODiag, LoggingLib, asstring, ArEventLog, AsTCP, snprintf, MpFile, MpServer, AsBrMath, MpAxis, MpRecipe, MpAlarmX, RandLib, SceneView, McPureVAx, SlFreeBase, arssl, powerlnk, asusb, asarlog, asarprof, dataobj, asmem, asio, aruser, asmath, MpRobotics, asepl
```

### Hardware
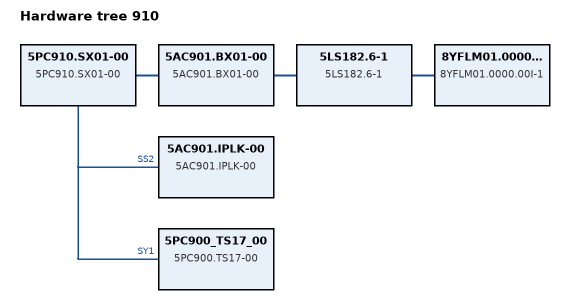
```
5AC901.BX01-00 : 5AC901.BX01-00 v1.1.0.0  [SY -> 5PC910.SX01-00.SY3]
5AC901.IPLK-00 : 5AC901.IPLK-00 v1.7.1.0  [SS -> 5PC910.SX01-00.SS2]
  Connector IF1:
    EplNatSubnet = 192.168.102.0
    Channel1
    ChannelID1 = McAcpBroadcast
    ChannelType1 = OCTET[96]
5LS182.6-1 : 5LS182.6-1 v1.3.1.0  [SL -> 5AC901.BX01-00.SL1]
  Connector IF1:
    CycleTime = 1000
5PC900_TS17_00 : 5PC900.TS17-00 v2.1.0.0  [SY -> 5PC910.SX01-00.SY1]
  ConfigurationID = OnsiteDemo_910
  UserPartitionSize = 10
  UserRamDevice = PCI.1.LS182.SRAM
  UserRamSize = 500000
  RemMemDevice = PCI.1.LS182.SRAM
  RemMemSize = 10000
  RemanentGlobalPvSize = 1000
  TimerDeviceType = EPLX2X
  TimerDevice = 5LS182.6-1.IF1
  Cyclic1Duration = 1000
  Cyclic1Tolerance = 0
  Cyclic2Duration = 5000
  Cyclic8Duration = 2000
  FileDevice1
  FileDeviceName1 = 6DMacro
  FileDevicePath1 = F:\Macros
  FileDevice2
  FileDeviceName2 = CNC_PrgDir
  FileDevicePath2 = F:/Programs/
  FileDevice3
  FileDeviceName3 = Recipe
  FileDevicePath3 = F:/Recipes/
  FileDevice4
  FileDeviceName4 = TeachFileDev
  FileDevicePath4 = F:/Teach/
  FileDevice5
  FileDeviceName5 = SvMovies
  FileDevicePath5 = F:/SvMovie
  FtpUser1
  FtpUsername1 = user  // user
  FtpUserPassword1 = uWQ3MCiALScWh+25zsAuoOpgOm0XOB8wRCPxpHYIgE4=  // user
  FtpUserSalt1 = pXahafUb
  FTPAccessRight1 = 0
  FTPdevice1 = ALL
  ActivateOpcUa = 1
  OpcUaPort = 4841
  OpcUaInformationModels_PV_Version = 2
5PC910.SX01-00 : 5PC910.SX01-00 v2.1.0.0
  Connector IF1:
    AssignedOperatingSystem = ARemb
  Connector IF3:
    AssignedOperatingSystem = ARemb
    ActivateDevice = 1
    Mode = Manual
    InternetAddress = 192.168.2.81
    SubnetMask = 255.255.255.0
    ActivateSnmp = 2
  Connector IF4:
    AssignedOperatingSystem = ARemb
    ActivateDevice = 1
  Connector IF5:
    AssignedOperatingSystem = ARemb
  Connector IF6:
    AssignedOperatingSystem = ARemb
  Connector IF7:
    AssignedOperatingSystem = ARemb
  Connector IF8:
    AssignedOperatingSystem = ARemb
  Connector IF9:
    AssignedOperatingSystem = ARemb
8YFLM01.0000.00I-1 : 8YFLM01.0000.00I-1 v0.0.0.1  [PLK1 -> 5LS182.6-1.IF1 (NodeNumber=1) [Cable Type=PowerlinkCable, Length=10, Version=1.0.0.3]]
  Supervision = off
```

### IoMap.iom - 5PC900_TS17_00/IoMap.iom
```iecst
VAR_CONFIG
	Cyclic#1.::FBin[0] AT %IW."8YFLM01.0000.00I-1".EPL_FB_IN_0_I2007_S01;
	Cyclic#1.::FBin[1] AT %IW."8YFLM01.0000.00I-1".EPL_FB_IN_1_I2007_S02;
	Cyclic#1.::FBin[10] AT %IW."8YFLM01.0000.00I-1".EPL_FB_IN_10_I2007_S0B;
	Cyclic#1.::FBin[100] AT %IW."8YFLM01.0000.00I-1".EPL_FB_IN_100_I2007_S65;
	Cyclic#1.::FBin[101] AT %IW."8YFLM01.0000.00I-1".EPL_FB_IN_101_I2007_S66;
	Cyclic#1.::FBin[102] AT %IW."8YFLM01.0000.00I-1".EPL_FB_IN_102_I2007_S67;
	Cyclic#1.::FBin[103] AT %IW."8YFLM01.0000.00I-1".EPL_FB_IN_103_I2007_S68;
	Cyclic#1.::FBin[104] AT %IW."8YFLM01.0000.00I-1".EPL_FB_IN_104_I2007_S69;
	Cyclic#1.::FBin[105] AT %IW."8YFLM01.0000.00I-1".EPL_FB_IN_105_I2007_S6A;
	Cyclic#1.::FBin[106] AT %IW."8YFLM01.0000.00I-1".EPL_FB_IN_106_I2007_S6B;
	Cyclic#1.::FBin[107] AT %IW."8YFLM01.0000.00I-1".EPL_FB_IN_107_I2007_S6C;
	Cyclic#1.::FBin[108] AT %IW."8YFLM01.0000.00I-1".EPL_FB_IN_108_I2007_S6D;
	Cyclic#1.::FBin[109] AT %IW."8YFLM01.0000.00I-1".EPL_FB_IN_109_I2007_S6E;
	Cyclic#1.::FBin[11] AT %IW."8YFLM01.0000.00I-1".EPL_FB_IN_11_I2007_S0C;
	Cyclic#1.::FBin[110] AT %IW."8YFLM01.0000.00I-1".EPL_FB_IN_110_I2007_S6F;
	Cyclic#1.::FBin[111] AT %IW."8YFLM01.0000.00I-1".EPL_FB_IN_111_I2007_S70;
	Cyclic#1.::FBin[112] AT %IW."8YFLM01.0000.00I-1".EPL_FB_IN_112_I2007_S71;
	Cyclic#1.::FBin[113] AT %IW."8YFLM01.0000.00I-1".EPL_FB_IN_113_I2007_S72;
	Cyclic#1.::FBin[114] AT %IW."8YFLM01.0000.00I-1".EPL_FB_IN_114_I2007_S73;
	Cyclic#1.::FBin[115] AT %IW."8YFLM01.0000.00I-1".EPL_FB_IN_115_I2007_S74;
	Cyclic#1.::FBin[116] AT %IW."8YFLM01.0000.00I-1".EPL_FB_IN_116_I2007_S75;
	Cyclic#1.::FBin[117] AT %IW."8YFLM01.0000.00I-1".EPL_FB_IN_117_I2007_S76;
	Cyclic#1.::FBin[118] AT %IW."8YFLM01.0000.00I-1".EPL_FB_IN_118_I2007_S77;
	Cyclic#1.::FBin[119] AT %IW."8YFLM01.0000.00I-1".EPL_FB_IN_119_I2007_S78;
	Cyclic#1.::FBin[12] AT %IW."8YFLM01.0000.00I-1".EPL_FB_IN_12_I2007_S0D;
	Cyclic#1.::FBin[120] AT %IW."8YFLM01.0000.00I-1".EPL_FB_IN_120_I2007_S79;
	Cyclic#1.::FBin[121] AT %IW."8YFLM01.0000.00I-1".EPL_FB_IN_121_I2007_S7A;
	Cyclic#1.::FBin[122] AT %IW."8YFLM01.0000.00I-1".EPL_FB_IN_122_I2007_S7B;
	Cyclic#1.::FBin[123] AT %IW."8YFLM01.0000.00I-1".EPL_FB_IN_123_I2007_S7C;
	Cyclic#1.::FBin[124] AT %IW."8YFLM01.0000.00I-1".EPL_FB_IN_124_I2007_S7D;
	Cyclic#1.::FBin[125] AT %IW."8YFLM01.0000.00I-1".EPL_FB_IN_125_I2007_S7E;
	Cyclic#1.::FBin[126] AT %IW."8YFLM01.0000.00I-1".EPL_FB_IN_126_I2007_S7F;
	Cyclic#1.::FBin[127] AT %IW."8YFLM01.0000.00I-1".EPL_FB_IN_127_I2007_S80;
	Cyclic#1.::FBin[128] AT %IW."8YFLM01.0000.00I-1".EPL_FB_IN_128_I2007_S81;
	Cyclic#1.::FBin[129] AT %IW."8YFLM01.0000.00I-1".EPL_FB_IN_129_I2007_S82;
	Cyclic#1.::FBin[13] AT %IW."8YFLM01.0000.00I-1".EPL_FB_IN_13_I2007_S0E;
	Cyclic#1.::FBin[130] AT %IW."8YFLM01.0000.00I-1".EPL_FB_IN_130_I2007_S83;
	Cyclic#1.::FBin[131] AT %IW."8YFLM01.0000.00I-1".EPL_FB_IN_131_I2007_S84;
	Cyclic#1.::FBin[132] AT %IW."8YFLM01.0000.00I-1".EPL_FB_IN_132_I2007_S85;
	Cyclic#1.::FBin[133] AT %IW."8YFLM01.0000.00I-1".EPL_FB_IN_133_I2007_S86;
	Cyclic#1.::FBin[134] AT %IW."8YFLM01.0000.00I-1".EPL_FB_IN_134_I2007_S87;
	Cyclic#1.::FBin[135] AT %IW."8YFLM01.0000.00I-1".EPL_FB_IN_135_I2007_S88;
	Cyclic#1.::FBin[136] AT %IW."8YFLM01.0000.00I-1".EPL_FB_IN_136_I2007_S89;
	Cyclic#1.::FBin[137] AT %IW."8YFLM01.0000.00I-1".EPL_FB_IN_137_I2007_S8A;
	Cyclic#1.::FBin[138] AT %IW."8YFLM01.0000.00I-1".EPL_FB_IN_138_I2007_S8B;
	Cyclic#1.::FBin[139] AT %IW."8YFLM01.0000.00I-1".EPL_FB_IN_139_I2007_S8C;
	Cyclic#1.::FBin[14] AT %IW."8YFLM01.0000.00I-1".EPL_FB_IN_14_I2007_S0F;
	Cyclic#1.::FBin[140] AT %IW."8YFLM01.0000.00I-1".EPL_FB_IN_140_I2007_S8D;
	Cyclic#1.::FBin[141] AT %IW."8YFLM01.0000.00I-1".EPL_FB_IN_141_I2007_S8E;
	Cyclic#1.::FBin[142] AT %IW."8YFLM01.0000.00I-1".EPL_FB_IN_142_I2007_S8F;
	Cyclic#1.::FBin[143] AT %IW."8YFLM01.0000.00I-1".EPL_FB_IN_143_I2007_S90;
	Cyclic#1.::FBin[144] AT %IW."8YFLM01.0000.00I-1".EPL_FB_IN_144_I2007_S91;
	Cyclic#1.::FBin[145] AT %IW."8YFLM01.0000.00I-1".EPL_FB_IN_145_I2007_S92;
	Cyclic#1.::FBin[146] AT %IW."8YFLM01.0000.00I-1".EPL_FB_IN_146_I2007_S93;
	Cyclic#1.::FBin[147] AT %IW."8YFLM01.0000.00I-1".EPL_FB_IN_147_I2007_S94;
	Cyclic#1.::FBin[148] AT %IW."8YFLM01.0000.00I-1".EPL_FB_IN_148_I2007_S95;
	Cyclic#1.::FBin[149] AT %IW."8YFLM01.0000.00I-1".EPL_FB_IN_149_I2007_S96;
	Cyclic#1.::FBin[15] AT %IW."8YFLM01.0000.00I-1".EPL_FB_IN_15_I2007_S10;
	Cyclic#1.::FBin[150] AT %IW."8YFLM01.0000.00I-1".EPL_FB_IN_150_I2007_S97;
	Cyclic#1.::FBin[151] AT %IW."8YFLM01.0000.00I-1".EPL_FB_IN_151_I2007_S98;
	Cyclic#1.::FBin[152] AT %IW."8YFLM01.0000.00I-1".EPL_FB_IN_152_I2007_S99;
	Cyclic#1.::FBin[153] AT %IW."8YFLM01.0000.00I-1".EPL_FB_IN_153_I2007_S9A;
	Cyclic#1.::FBin[154] AT %IW."8YFLM01.0000.00I-1".EPL_FB_IN_154_I2007_S9B;
	Cyclic#1.::FBin[155] AT %IW."8YFLM01.0000.00I-1".EPL_FB_IN_155_I2007_S9C;
	Cyclic#1.::FBin[156] AT %IW."8YFLM01.0000.00I-1".EPL_FB_IN_156_I2007_S9D;
	Cyclic#1.::FBin[157] AT %IW."8YFLM01.0000.00I-1".EPL_FB_IN_157_I2007_S9E;
	Cyclic#1.::FBin[158] AT %IW."8YFLM01.0000.00I-1".EPL_FB_IN_158_I2007_S9F;
	Cyclic#1.::FBin[159] AT %IW."8YFLM01.0000.00I-1".EPL_FB_IN_159_I2007_SA0;
	Cyclic#1.::FBin[16] AT %IW."8YFLM01.0000.00I-1".EPL_FB_IN_16_I2007_S11;
	Cyclic#1.::FBin[160] AT %IW."8YFLM01.0000.00I-1".EPL_FB_IN_160_I2007_SA1;
	Cyclic#1.::FBin[161] AT %IW."8YFLM01.0000.00I-1".EPL_FB_IN_161_I2007_SA2;
	Cyclic#1.::FBin[162] AT %IW."8YFLM01.0000.00I-1".EPL_FB_IN_162_I2007_SA3;
	Cyclic#1.::FBin[163] AT %IW."8YFLM01.0000.00I-1".EPL_FB_IN_163_I2007_SA4;
	Cyclic#1.::FBin[164] AT %IW."8YFLM01.0000.00I-1".EPL_FB_IN_164_I2007_SA5;
	Cyclic#1.::FBin[165] AT %IW."8YFLM01.0000.00I-1".EPL_FB_IN_165_I2007_SA6;
	Cyclic#1.::FBin[166] AT %IW."8YFLM01.0000.00I-1".EPL_FB_IN_166_I2007_SA7;
	Cyclic#1.::FBin[167] AT %IW."8YFLM01.0000.00I-1".EPL_FB_IN_167_I2007_SA8;
	Cyclic#1.::FBin[168] AT %IW."8YFLM01.0000.00I-1".EPL_FB_IN_168_I2007_SA9;
	Cyclic#1.::FBin[169] AT %IW."8YFLM01.0000.00I-1".EPL_FB_IN_169_I2007_SAA;
	Cyclic#1.::FBin[17] AT %IW."8YFLM01.0000.00I-1".EPL_FB_IN_17_I2007_S12;
	Cyclic#1.::FBin[170] AT %IW."8YFLM01.0000.00I-1".EPL_FB_IN_170_I2007_SAB;
	Cyclic#1.::FBin[171] AT %IW."8YFLM01.0000.00I-1".EPL_FB_IN_171_I2007_SAC;
	Cyclic#1.::FBin[172] AT %IW."8YFLM01.0000.00I-1".EPL_FB_IN_172_I2007_SAD;
	Cyclic#1.::FBin[173] AT %IW."8YFLM01.0000.00I-1".EPL_FB_IN_173_I2007_SAE;
	Cyclic#1.::FBin[174] AT %IW."8YFLM01.0000.00I-1".EPL_FB_IN_174_I2007_SAF;
	Cyclic#1.::FBin[175] AT %IW."8YFLM01.0000.00I-1".EPL_FB_IN_175_I2007_SB0;
	Cyclic#1.::FBin[176] AT %IW."8YFLM01.0000.00I-1".EPL_FB_IN_176_I2007_SB1;
	Cyclic#1.::FBin[177] AT %IW."8YFLM01.0000.00I-1".EPL_FB_IN_177_I2007_SB2;
	Cyclic#1.::FBin[178] AT %IW."8YFLM01.0000.00I-1".EPL_FB_IN_178_I2007_SB3;
	Cyclic#1.::FBin[179] AT %IW."8YFLM01.0000.00I-1".EPL_FB_IN_179_I2007_SB4;
	Cyclic#1.::FBin[18] AT %IW."8YFLM01.0000.00I-1".EPL_FB_IN_18_I2007_S13;
	Cyclic#1.::FBin[180] AT %IW."8YFLM01.0000.00I-1".EPL_FB_IN_180_I2007_SB5;
	Cyclic#1.::FBin[181] AT %IW."8YFLM01.0000.00I-1".EPL_FB_IN_181_I2007_SB6;
	Cyclic#1.::FBin[182] AT %IW."8YFLM01.0000.00I-1".EPL_FB_IN_182_I2007_SB7;
	Cyclic#1.::FBin[183] AT %IW."8YFLM01.0000.00I-1".EPL_FB_IN_183_I2007_SB8;
	Cyclic#1.::FBin[184] AT %IW."8YFLM01.0000.00I-1".EPL_FB_IN_184_I2007_SB9;
	Cyclic#1.::FBin[185] AT %IW."8YFLM01.0000.00I-1".EPL_FB_IN_185_I2007_SBA;
	Cyclic#1.::FBin[186] AT %IW."8YFLM01.0000.00I-1".EPL_FB_IN_186_I2007_SBB;
	Cyclic#1.::FBin[187] AT %IW."8YFLM01.0000.00I-1".EPL_FB_IN_187_I2007_SBC;
	Cyclic#1.::FBin[188] AT %IW."8YFLM01.0000.00I-1".EPL_FB_IN_188_I2007_SBD;
	Cyclic#1.::FBin[189] AT %IW."8YFLM01.0000.00I-1".EPL_FB_IN_189_I2007_SBE;
	Cyclic#1.::FBin[19] AT %IW."8YFLM01.0000.00I-1".EPL_FB_IN_19_I2007_S14;
	Cyclic#1.::FBin[190] AT %IW."8YFLM01.0000.00I-1".EPL_FB_IN_190_I2007_SBF;
	Cyclic#1.::FBin[191] AT %IW."8YFLM01.0000.00I-1".EPL_FB_IN_191_I2007_SC0;
	Cyclic#1.::FBin[192] AT %IW."8YFLM01.0000.00I-1".EPL_FB_IN_192_I2007_SC1;
	Cyclic#1.::FBin[193] AT %IW."8YFLM01.0000.00I-1".EPL_FB_IN_193_I2007_SC2;
	Cyclic#1.::FBin[194] AT %IW."8YFLM01.0000.00I-1".EPL_FB_IN_194_I2007_SC3;
	Cyclic#1.::FBin[195] AT %IW."8YFLM01.0000.00I-1".EPL_FB_IN_195_I2007_SC4;
	Cyclic#1.::FBin[196] AT %IW."8YFLM01.0000.00I-1".EPL_FB_IN_196_I2007_SC5;
	Cyclic#1.::FBin[197] AT %IW."8YFLM01.0000.00I-1".EPL_FB_IN_197_I2007_SC6;
	Cyclic#1.::FBin[198] AT %IW."8YFLM01.0000.00I-1".EPL_FB_IN_198_I2007_SC7;
	Cyclic#1.::FBin[199] AT %IW."8YFLM01.0000.00I-1".EPL_FB_IN_199_I2007_SC8;
	Cyclic#1.::FBin[2] AT %IW."8YFLM01.0000.00I-1".EPL_FB_IN_2_I2007_S03;
	Cyclic#1.::FBin[20] AT %IW."8YFLM01.0000.00I-1".EPL_FB_IN_20_I2007_S15;
	Cyclic#1.::FBin[21] AT %IW."8YFLM01.0000.00I-1".EPL_FB_IN_21_I2007_S16;
	Cyclic#1.::FBin[22] AT %IW."8YFLM01.0000.00I-1".EPL_FB_IN_22_I2007_S17;
	Cyclic#1.::FBin[23] AT %IW."8YFLM01.0000.00I-1".EPL_FB_IN_23_I2007_S18;
	Cyclic#1.::FBin[24] AT %IW."8YFLM01.0000.00I-1".EPL_FB_IN_24_I2007_S19;
	Cyclic#1.::FBin[25] AT %IW."8YFLM01.0000.00I-1".EPL_FB_IN_25_I2007_S1A;
	Cyclic#1.::FBin[26] AT %IW."8YFLM01.0000.00I-1".EPL_FB_IN_26_I2007_S1B;
	Cyclic#1.::FBin[27] AT %IW."8YFLM01.0000.00I-1".EPL_FB_IN_27_I2007_S1C;
	Cyclic#1.::FBin[28] AT %IW."8YFLM01.0000.00I-1".EPL_FB_IN_28_I2007_S1D;
	Cyclic#1.::FBin[29] AT %IW."8YFLM01.0000.00I-1".EPL_FB_IN_29_I2007_S1E;
	Cyclic#1.::FBin[3] AT %IW."8YFLM01.0000.00I-1".EPL_FB_IN_3_I2007_S04;
	Cyclic#1.::FBin[30] AT %IW."8YFLM01.0000.00I-1".EPL_FB_IN_30_I2007_S1F;
	Cyclic#1.::FBin[31] AT %IW."8YFLM01.0000.00I-1".EPL_FB_IN_31_I2007_S20;
	Cyclic#1.::FBin[32] AT %IW."8YFLM01.0000.00I-1".EPL_FB_IN_32_I2007_S21;
	Cyclic#1.::FBin[33] AT %IW."8YFLM01.0000.00I-1".EPL_FB_IN_33_I2007_S22;
	Cyclic#1.::FBin[34] AT %IW."8YFLM01.0000.00I-1".EPL_FB_IN_34_I2007_S23;
	Cyclic#1.::FBin[35] AT %IW."8YFLM01.0000.00I-1".EPL_FB_IN_35_I2007_S24;
	Cyclic#1.::FBin[36] AT %IW."8YFLM01.0000.00I-1".EPL_FB_IN_36_I2007_S25;
	Cyclic#1.::FBin[37] AT %IW."8YFLM01.0000.00I-1".EPL_FB_IN_37_I2007_S26;
	Cyclic#1.::FBin[38] AT %IW."8YFLM01.0000.00I-1".EPL_FB_IN_38_I2007_S27;
	Cyclic#1.::FBin[39] AT %IW."8YFLM01.0000.00I-1".EPL_FB_IN_39_I2007_S28;
	Cyclic#1.::FBin[4] AT %IW."8YFLM01.0000.00I-1".EPL_FB_IN_4_I2007_S05;
	Cyclic#1.::FBin[40] AT %IW."8YFLM01.0000.00I-1".EPL_FB_IN_40_I2007_S29;
	Cyclic#1.::FBin[41] AT %IW."8YFLM01.0000.00I-1".EPL_FB_IN_41_I2007_S2A;
	Cyclic#1.::FBin[42] AT %IW."8YFLM01.0000.00I-1".EPL_FB_IN_42_I2007_S2B;
	Cyclic#1.::FBin[43] AT %IW."8YFLM01.0000.00I-1".EPL_FB_IN_43_I2007_S2C;
	Cyclic#1.::FBin[44] AT %IW."8YFLM01.0000.00I-1".EPL_FB_IN_44_I2007_S2D;
	Cyclic#1.::FBin[45] AT %IW."8YFLM01.0000.00I-1".EPL_FB_IN_45_I2007_S2E;
	Cyclic#1.::FBin[46] AT %IW."8YFLM01.0000.00I-1".EPL_FB_IN_46_I2007_S2F;
	Cyclic#1.::FBin[47] AT %IW."8YFLM01.0000.00I-1".EPL_FB_IN_47_I2007_S30;
	Cyclic#1.::FBin[48] AT %IW."8YFLM01.0000.00I-1".EPL_FB_IN_48_I2007_S31;
	Cyclic#1.::FBin[49] AT %IW."8YFLM01.0000.00I-1".EPL_FB_IN_49_I2007_S32;
	Cyclic#1.::FBin[5] AT %IW."8YFLM01.0000.00I-1".EPL_FB_IN_5_I2007_S06;
	Cyclic#1.::FBin[50] AT %IW."8YFLM01.0000.00I-1".EPL_FB_IN_50_I2007_S33;
	Cyclic#1.::FBin[51] AT %IW."8YFLM01.0000.00I-1".EPL_FB_IN_51_I2007_S34;
	Cyclic#1.::FBin[52] AT %IW."8YFLM01.0000.00I-1".EPL_FB_IN_52_I2007_S35;
	Cyclic#1.::FBin[53] AT %IW."8YFLM01.0000.00I-1".EPL_FB_IN_53_I2007_S36;
	Cyclic#1.::FBin[54] AT %IW."8YFLM01.0000.00I-1".EPL_FB_IN_54_I2007_S37;
	Cyclic#1.::FBin[55] AT %IW."8YFLM01.0000.00I-1".EPL_FB_IN_55_I2007_S38;
	Cyclic#1.::FBin[56] AT %IW."8YFLM01.0000.00I-1".EPL_FB_IN_56_I2007_S39;
	Cyclic#1.::FBin[57] AT %IW."8YFLM01.0000.00I-1".EPL_FB_IN_57_I2007_S3A;
	Cyclic#1.::FBin[58] AT %IW."8YFLM01.0000.00I-1".EPL_FB_IN_58_I2007_S3B;
	Cyclic#1.::FBin[59] AT %IW."8YFLM01.0000.00I-1".EPL_FB_IN_59_I2007_S3C;
	Cyclic#1.::FBin[6] AT %IW."8YFLM01.0000.00I-1".EPL_FB_IN_6_I2007_S07;
	Cyclic#1.::FBin[60] AT %IW."8YFLM01.0000.00I-1".EPL_FB_IN_60_I2007_S3D;
	Cyclic#1.::FBin[61] AT %IW."8YFLM01.0000.00I-1".EPL_FB_IN_61_I2007_S3E;
	Cyclic#1.::FBin[62] AT %IW."8YFLM01.0000.00I-1".EPL_FB_IN_62_I2007_S3F;
	Cyclic#1.::FBin[63] AT %IW."8YFLM01.0000.00I-1".EPL_FB_IN_63_I2007_S40;
	Cyclic#1.::FBin[64] AT %IW."8YFLM01.0000.00I-1".EPL_FB_IN_64_I2007_S41;
	Cyclic#1.::FBin[65] AT %IW."8YFLM01.0000.00I-1".EPL_FB_IN_65_I2007_S42;
	Cyclic#1.::FBin[66] AT %IW."8YFLM01.0000.00I-1".EPL_FB_IN_66_I2007_S43;
	Cyclic#1.::FBin[67] AT %IW."8YFLM01.0000.00I-1".EPL_FB_IN_67_I2007_S44;
	Cyclic#1.::FBin[68] AT %IW."8YFLM01.0000.00I-1".EPL_FB_IN_68_I2007_S45;
	Cyclic#1.::FBin[69] AT %IW."8YFLM01.0000.00I-1".EPL_FB_IN_69_I2007_S46;
	Cyclic#1.::FBin[7] AT %IW."8YFLM01.0000.00I-1".EPL_FB_IN_7_I2007_S08;
	Cyclic#1.::FBin[70] AT %IW."8YFLM01.0000.00I-1".EPL_FB_IN_70_I2007_S47;
	Cyclic#1.::FBin[71] AT %IW."8YFLM01.0000.00I-1".EPL_FB_IN_71_I2007_S48;
	Cyclic#1.::FBin[72] AT %IW."8YFLM01.0000.00I-1".EPL_FB_IN_72_I2007_S49;
	Cyclic#1.::FBin[73] AT %IW."8YFLM01.0000.00I-1".EPL_FB_IN_73_I2007_S4A;
	Cyclic#1.::FBin[74] AT %IW."8YFLM01.0000.00I-1".EPL_FB_IN_74_I2007_S4B;
	Cyclic#1.::FBin[75] AT %IW."8YFLM01.0000.00I-1".EPL_FB_IN_75_I2007_S4C;
	Cyclic#1.::FBin[76] AT %IW."8YFLM01.0000.00I-1".EPL_FB_IN_76_I2007_S4D;
	Cyclic#1.::FBin[77] AT %IW."8YFLM01.0000.00I-1".EPL_FB_IN_77_I2007_S4E;
	Cyclic#1.::FBin[78] AT %IW."8YFLM01.0000.00I-1".EPL_FB_IN_78_I2007_S4F;
	Cyclic#1.::FBin[79] AT %IW."8YFLM01.0000.00I-1".EPL_FB_IN_79_I2007_S50;
	Cyclic#1.::FBin[8] AT %IW."8YFLM01.0000.00I-1".EPL_FB_IN_8_I2007_S09;
	Cyclic#1.::FBin[80] AT %IW."8YFLM01.0000.00I-1".EPL_FB_IN_80_I2007_S51;
	Cyclic#1.::FBin[81] AT %IW."8YFLM01.0000.00I-1".EPL_FB_IN_81_I2007_S52;
	Cyclic#1.::FBin[82] AT %IW."8YFLM01.0000.00I-1".EPL_FB_IN_82_I2007_S53;
	Cyclic#1.::FBin[83] AT %IW."8YFLM01.0000.00I-1".EPL_FB_IN_83_I2007_S54;
	Cyclic#1.::FBin[84] AT %IW."8YFLM01.0000.00I-1".EPL_FB_IN_84_I2007_S55;
	Cyclic#1.::FBin[85] AT %IW."8YFLM01.0000.00I-1".EPL_FB_IN_85_I2007_S56;
	Cyclic#1.::FBin[86] AT %IW."8YFLM01.0000.00I-1".EPL_FB_IN_86_I2007_S57;
	Cyclic#1.::FBin[87] AT %IW."8YFLM01.0000.00I-1".EPL_FB_IN_87_I2007_S58;
	Cyclic#1.::FBin[88] AT %IW."8YFLM01.0000.00I-1".EPL_FB_IN_88_I2007_S59;
	Cyclic#1.::FBin[89] AT %IW."8YFLM01.0000.00I-1".EPL_FB_IN_89_I2007_S5A;
	Cyclic#1.::FBin[9] AT %IW."8YFLM01.0000.00I-1".EPL_FB_IN_9_I2007_S0A;
	Cyclic#1.::FBin[90] AT %IW."8YFLM01.0000.00I-1".EPL_FB_IN_90_I2007_S5B;
	Cyclic#1.::FBin[91] AT %IW."8YFLM01.0000.00I-1".EPL_FB_IN_91_I2007_S5C;
	Cyclic#1.::FBin[92] AT %IW."8YFLM01.0000.00I-1".EPL_FB_IN_92_I2007_S5D;
	Cyclic#1.::FBin[93] AT %IW."8YFLM01.0000.00I-1".EPL_FB_IN_93_I2007_S5E;
	Cyclic#1.::FBin[94] AT %IW."8YFLM01.0000.00I-1".EPL_FB_IN_94_I2007_S5F;
	Cyclic#1.::FBin[95] AT %IW."8YFLM01.0000.00I-1".EPL_FB_IN_95_I2007_S60;
	Cyclic#1.::FBin[96] AT %IW."8YFLM01.0000.00I-1".EPL_FB_IN_96_I2007_S61;
	Cyclic#1.::FBin[97] AT %IW."8YFLM01.0000.00I-1".EPL_FB_IN_97_I2007_S62;
	Cyclic#1.::FBin[98] AT %IW."8YFLM01.0000.00I-1".EPL_FB_IN_98_I2007_S63;
	Cyclic#1.::FBin[99] AT %IW."8YFLM01.0000.00I-1".EPL_FB_IN_99_I2007_S64;
	Cyclic#1.::FBout[0] AT %QW."8YFLM01.0000.00I-1".EPL_FB_OUT_0_I2008_S01Out;
	Cyclic#1.::FBout[1] AT %QW."8YFLM01.0000.00I-1".EPL_FB_OUT_1_I2008_S02Out;
	Cyclic#1.::FBout[10] AT %QW."8YFLM01.0000.00I-1".EPL_FB_OUT_10_I2008_S0BOut;
	Cyclic#1.::FBout[100] AT %QW."8YFLM01.0000.00I-1".EPL_FB_OUT_100_I2008_S65Out;
	Cyclic#1.::FBout[101] AT %QW."8YFLM01.0000.00I-1".EPL_FB_OUT_101_I2008_S66Out;
	Cyclic#1.::FBout[102] AT %QW."8YFLM01.0000.00I-1".EPL_FB_OUT_102_I2008_S67Out;
	Cyclic#1.::FBout[103] AT %QW."8YFLM01.0000.00I-1".EPL_FB_OUT_103_I2008_S68Out;
	Cyclic#1.::FBout[104] AT %QW."8YFLM01.0000.00I-1".EPL_FB_OUT_104_I2008_S69Out;
	Cyclic#1.::FBout[105] AT %QW."8YFLM01.0000.00I-1".EPL_FB_OUT_105_I2008_S6AOut;
	Cyclic#1.::FBout[106] AT %QW."8YFLM01.0000.00I-1".EPL_FB_OUT_106_I2008_S6BOut;
	Cyclic#1.::FBout[107] AT %QW."8YFLM01.0000.00I-1".EPL_FB_OUT_107_I2008_S6COut;
	Cyclic#1.::FBout[108] AT %QW."8YFLM01.0000.00I-1".EPL_FB_OUT_108_I2008_S6DOut;
	Cyclic#1.::FBout[109] AT %QW."8YFLM01.0000.00I-1".EPL_FB_OUT_109_I2008_S6EOut;
	Cyclic#1.::FBout[11] AT %QW."8YFLM01.0000.00I-1".EPL_FB_OUT_11_I2008_S0COut;
	Cyclic#1.::FBout[110] AT %QW."8YFLM01.0000.00I-1".EPL_FB_OUT_110_I2008_S6FOut;
	Cyclic#1.::FBout[111] AT %QW."8YFLM01.0000.00I-1".EPL_FB_OUT_111_I2008_S70Out;
	Cyclic#1.::FBout[112] AT %QW."8YFLM01.0000.00I-1".EPL_FB_OUT_112_I2008_S71Out;
	Cyclic#1.::FBout[113] AT %QW."8YFLM01.0000.00I-1".EPL_FB_OUT_113_I2008_S72Out;
	Cyclic#1.::FBout[114] AT %QW."8YFLM01.0000.00I-1".EPL_FB_OUT_114_I2008_S73Out;
	Cyclic#1.::FBout[115] AT %QW."8YFLM01.0000.00I-1".EPL_FB_OUT_115_I2008_S74Out;
	Cyclic#1.::FBout[116] AT %QW."8YFLM01.0000.00I-1".EPL_FB_OUT_116_I2008_S75Out;
	Cyclic#1.::FBout[117] AT %QW."8YFLM01.0000.00I-1".EPL_FB_OUT_117_I2008_S76Out;
	Cyclic#1.::FBout[118] AT %QW."8YFLM01.0000.00I-1".EPL_FB_OUT_118_I2008_S77Out;
	Cyclic#1.::FBout[119] AT %QW."8YFLM01.0000.00I-1".EPL_FB_OUT_119_I2008_S78Out;
	Cyclic#1.::FBout[12] AT %QW."8YFLM01.0000.00I-1".EPL_FB_OUT_12_I2008_S0DOut;
	Cyclic#1.::FBout[120] AT %QW."8YFLM01.0000.00I-1".EPL_FB_OUT_120_I2008_S79Out;
	Cyclic#1.::FBout[121] AT %QW."8YFLM01.0000.00I-1".EPL_FB_OUT_121_I2008_S7AOut;
	Cyclic#1.::FBout[122] AT %QW."8YFLM01.0000.00I-1".EPL_FB_OUT_122_I2008_S7BOut;
	Cyclic#1.::FBout[123] AT %QW."8YFLM01.0000.00I-1".EPL_FB_OUT_123_I2008_S7COut;
	Cyclic#1.::FBout[124] AT %QW."8YFLM01.0000.00I-1".EPL_FB_OUT_124_I2008_S7DOut;
	Cyclic#1.::FBout[125] AT %QW."8YFLM01.0000.00I-1".EPL_FB_OUT_125_I2008_S7EOut;
	Cyclic#1.::FBout[126] AT %QW."8YFLM01.0000.00I-1".EPL_FB_OUT_126_I2008_S7FOut;
	Cyclic#1.::FBout[127] AT %QW."8YFLM01.0000.00I-1".EPL_FB_OUT_127_I2008_S80Out;
	Cyclic#1.::FBout[128] AT %QW."8YFLM01.0000.00I-1".EPL_FB_OUT_128_I2008_S81Out;
	Cyclic#1.::FBout[129] AT %QW."8YFLM01.0000.00I-1".EPL_FB_OUT_129_I2008_S82Out;
	Cyclic#1.::FBout[13] AT %QW."8YFLM01.0000.00I-1".EPL_FB_OUT_13_I2008_S0EOut;
	Cyclic#1.::FBout[130] AT %QW."8YFLM01.0000.00I-1".EPL_FB_OUT_130_I2008_S83Out;
	Cyclic#1.::FBout[131] AT %QW."8YFLM01.0000.00I-1".EPL_FB_OUT_131_I2008_S84Out;
	Cyclic#1.::FBout[132] AT %QW."8YFLM01.0000.00I-1".EPL_FB_OUT_132_I2008_S85Out;
	Cyclic#1.::FBout[133] AT %QW."8YFLM01.0000.00I-1".EPL_FB_OUT_133_I2008_S86Out;
	Cyclic#1.::FBout[134] AT %QW."8YFLM01.0000.00I-1".EPL_FB_OUT_134_I2008_S87Out;
	Cyclic#1.::FBout[135] AT %QW."8YFLM01.0000.00I-1".EPL_FB_OUT_135_I2008_S88Out;
	Cyclic#1.::FBout[136] AT %QW."8YFLM01.0000.00I-1".EPL_FB_OUT_136_I2008_S89Out;
	Cyclic#1.::FBout[137] AT %QW."8YFLM01.0000.00I-1".EPL_FB_OUT_137_I2008_S8AOut;
	Cyclic#1.::FBout[138] AT %QW."8YFLM01.0000.00I-1".EPL_FB_OUT_138_I2008_S8BOut;
	Cyclic#1.::FBout[139] AT %QW."8YFLM01.0000.00I-1".EPL_FB_OUT_139_I2008_S8COut;
	Cyclic#1.::FBout[14] AT %QW."8YFLM01.0000.00I-1".EPL_FB_OUT_14_I2008_S0FOut;
	Cyclic#1.::FBout[140] AT %QW."8YFLM01.0000.00I-1".EPL_FB_OUT_140_I2008_S8DOut;
	Cyclic#1.::FBout[141] AT %QW."8YFLM01.0000.00I-1".EPL_FB_OUT_141_I2008_S8EOut;
	Cyclic#1.::FBout[142] AT %QW."8YFLM01.0000.00I-1".EPL_FB_OUT_142_I2008_S8FOut;
	Cyclic#1.::FBout[143] AT %QW."8YFLM01.0000.00I-1".EPL_FB_OUT_143_I2008_S90Out;
	Cyclic#1.::FBout[144] AT %QW."8YFLM01.0000.00I-1".EPL_FB_OUT_144_I2008_S91Out;
	Cyclic#1.::FBout[145] AT %QW."8YFLM01.0000.00I-1".EPL_FB_OUT_145_I2008_S92Out;
	Cyclic#1.::FBout[146] AT %QW."8YFLM01.0000.00I-1".EPL_FB_OUT_146_I2008_S93Out;
	Cyclic#1.::FBout[147] AT %QW."8YFLM01.0000.00I-1".EPL_FB_OUT_147_I2008_S94Out;
	Cyclic#1.::FBout[148] AT %QW."8YFLM01.0000.00I-1".EPL_FB_OUT_148_I2008_S95Out;
	Cyclic#1.::FBout[149] AT %QW."8YFLM01.0000.00I-1".EPL_FB_OUT_149_I2008_S96Out;
	Cyclic#1.::FBout[15] AT %QW."8YFLM01.0000.00I-1".EPL_FB_OUT_15_I2008_S10Out;
	Cyclic#1.::FBout[150] AT %QW."8YFLM01.0000.00I-1".EPL_FB_OUT_150_I2008_S97Out;
	Cyclic#1.::FBout[151] AT %QW."8YFLM01.0000.00I-1".EPL_FB_OUT_151_I2008_S98Out;
	Cyclic#1.::FBout[152] AT %QW."8YFLM01.0000.00I-1".EPL_FB_OUT_152_I2008_S99Out;
	Cyclic#1.::FBout[153] AT %QW."8YFLM01.0000.00I-1".EPL_FB_OUT_153_I2008_S9AOut;
	Cyclic#1.::FBout[154] AT %QW."8YFLM01.0000.00I-1".EPL_FB_OUT_154_I2008_S9BOut;
	Cyclic#1.::FBout[155] AT %QW."8YFLM01.0000.00I-1".EPL_FB_OUT_155_I2008_S9COut;
	Cyclic#1.::FBout[156] AT %QW."8YFLM01.0000.00I-1".EPL_FB_OUT_156_I2008_S9DOut;
	Cyclic#1.::FBout[157] AT %QW."8YFLM01.0000.00I-1".EPL_FB_OUT_157_I2008_S9EOut;
	Cyclic#1.::FBout[158] AT %QW."8YFLM01.0000.00I-1".EPL_FB_OUT_158_I2008_S9FOut;
	Cyclic#1.::FBout[159] AT %QW."8YFLM01.0000.00I-1".EPL_FB_OUT_159_I2008_SA0Out;
	Cyclic#1.::FBout[16] AT %QW."8YFLM01.0000.00I-1".EPL_FB_OUT_16_I2008_S11Out;
	Cyclic#1.::FBout[160] AT %QW."8YFLM01.0000.00I-1".EPL_FB_OUT_160_I2008_SA1Out;
	Cyclic#1.::FBout[161] AT %QW."8YFLM01.0000.00I-1".EPL_FB_OUT_161_I2008_SA2Out;
	Cyclic#1.::FBout[162] AT %QW."8YFLM01.0000.00I-1".EPL_FB_OUT_162_I2008_SA3Out;
	Cyclic#1.::FBout[163] AT %QW."8YFLM01.0000.00I-1".EPL_FB_OUT_163_I2008_SA4Out;
	Cyclic#1.::FBout[164] AT %QW."8YFLM01.0000.00I-1".EPL_FB_OUT_164_I2008_SA5Out;
	Cyclic#1.::FBout[165] AT %QW."8YFLM01.0000.00I-1".EPL_FB_OUT_165_I2008_SA6Out;
	Cyclic#1.::FBout[166] AT %QW."8YFLM01.0000.00I-1".EPL_FB_OUT_166_I2008_SA7Out;
	Cyclic#1.::FBout[167] AT %QW."8YFLM01.0000.00I-1".EPL_FB_OUT_167_I2008_SA8Out;
	Cyclic#1.::FBout[168] AT %QW."8YFLM01.0000.00I-1".EPL_FB_OUT_168_I2008_SA9Out;
	Cyclic#1.::FBout[169] AT %QW."8YFLM01.0000.00I-1".EPL_FB_OUT_169_I2008_SAAOut;
	Cyclic#1.::FBout[17] AT %QW."8YFLM01.0000.00I-1".EPL_FB_OUT_17_I2008_S12Out;
	Cyclic#1.::FBout[170] AT %QW."8YFLM01.0000.00I-1".EPL_FB_OUT_170_I2008_SABOut;
	Cyclic#1.::FBout[171] AT %QW."8YFLM01.0000.00I-1".EPL_FB_OUT_171_I2008_SACOut;
	Cyclic#1.::FBout[172] AT %QW."8YFLM01.0000.00I-1".EPL_FB_OUT_172_I2008_SADOut;
	Cyclic#1.::FBout[173] AT %QW."8YFLM01.0000.00I-1".EPL_FB_OUT_173_I2008_SAEOut;
	Cyclic#1.::FBout[174] AT %QW."8YFLM01.0000.00I-1".EPL_FB_OUT_174_I2008_SAFOut;
	Cyclic#1.::FBout[175] AT %QW."8YFLM01.0000.00I-1".EPL_FB_OUT_175_I2008_SB0Out;
	Cyclic#1.::FBout[176] AT %QW."8YFLM01.0000.00I-1".EPL_FB_OUT_176_I2008_SB1Out;
	Cyclic#1.::FBout[177] AT %QW."8YFLM01.0000.00I-1".EPL_FB_OUT_177_I2008_SB2Out;
	Cyclic#1.::FBout[178] AT %QW."8YFLM01.0000.00I-1".EPL_FB_OUT_178_I2008_SB3Out;
	Cyclic#1.::FBout[179] AT %QW."8YFLM01.0000.00I-1".EPL_FB_OUT_179_I2008_SB4Out;
	Cyclic#1.::FBout[18] AT %QW."8YFLM01.0000.00I-1".EPL_FB_OUT_18_I2008_S13Out;
	Cyclic#1.::FBout[180] AT %QW."8YFLM01.0000.00I-1".EPL_FB_OUT_180_I2008_SB5Out;
	Cyclic#1.::FBout[181] AT %QW."8YFLM01.0000.00I-1".EPL_FB_OUT_181_I2008_SB6Out;
	Cyclic#1.::FBout[182] AT %QW."8YFLM01.0000.00I-1".EPL_FB_OUT_182_I2008_SB7Out;
	Cyclic#1.::FBout[183] AT %QW."8YFLM01.0000.00I-1".EPL_FB_OUT_183_I2008_SB8Out;
	Cyclic#1.::FBout[184] AT %QW."8YFLM01.0000.00I-1".EPL_FB_OUT_184_I2008_SB9Out;
	Cyclic#1.::FBout[185] AT %QW."8YFLM01.0000.00I-1".EPL_FB_OUT_185_I2008_SBAOut;
	Cyclic#1.::FBout[186] AT %QW."8YFLM01.0000.00I-1".EPL_FB_OUT_186_I2008_SBBOut;
	Cyclic#1.::FBout[187] AT %QW."8YFLM01.0000.00I-1".EPL_FB_OUT_187_I2008_SBCOut;
	Cyclic#1.::FBout[188] AT %QW."8YFLM01.0000.00I-1".EPL_FB_OUT_188_I2008_SBDOut;
	Cyclic#1.::FBout[189] AT %QW."8YFLM01.0000.00I-1".EPL_FB_OUT_189_I2008_SBEOut;
	Cyclic#1.::FBout[19] AT %QW."8YFLM01.0000.00I-1".EPL_FB_OUT_19_I2008_S14Out;
	Cyclic#1.::FBout[190] AT %QW."8YFLM01.0000.00I-1".EPL_FB_OUT_190_I2008_SBFOut;
	Cyclic#1.::FBout[191] AT %QW."8YFLM01.0000.00I-1".EPL_FB_OUT_191_I2008_SC0Out;
	Cyclic#1.::FBout[192] AT %QW."8YFLM01.0000.00I-1".EPL_FB_OUT_192_I2008_SC1Out;
	Cyclic#1.::FBout[193] AT %QW."8YFLM01.0000.00I-1".EPL_FB_OUT_193_I2008_SC2Out;
	Cyclic#1.::FBout[194] AT %QW."8YFLM01.0000.00I-1".EPL_FB_OUT_194_I2008_SC3Out;
	Cyclic#1.::FBout[195] AT %QW."8YFLM01.0000.00I-1".EPL_FB_OUT_195_I2008_SC4Out;
	Cyclic#1.::FBout[196] AT %QW."8YFLM01.0000.00I-1".EPL_FB_OUT_196_I2008_SC5Out;
	Cyclic#1.::FBout[197] AT %QW."8YFLM01.0000.00I-1".EPL_FB_OUT_197_I2008_SC6Out;
	Cyclic#1.::FBout[198] AT %QW."8YFLM01.0000.00I-1".EPL_FB_OUT_198_I2008_SC7Out;
	Cyclic#1.::FBout[199] AT %QW."8YFLM01.0000.00I-1".EPL_FB_OUT_199_I2008_SC8Out;
	Cyclic#1.::FBout[2] AT %QW."8YFLM01.0000.00I-1".EPL_FB_OUT_2_I2008_S03Out;
	Cyclic#1.::FBout[20] AT %QW."8YFLM01.0000.00I-1".EPL_FB_OUT_20_I2008_S15Out;
	Cyclic#1.::FBout[21] AT %QW."8YFLM01.0000.00I-1".EPL_FB_OUT_21_I2008_S16Out;
	Cyclic#1.::FBout[22] AT %QW."8YFLM01.0000.00I-1".EPL_FB_OUT_22_I2008_S17Out;
	Cyclic#1.::FBout[23] AT %QW."8YFLM01.0000.00I-1".EPL_FB_OUT_23_I2008_S18Out;
	Cyclic#1.::FBout[24] AT %QW."8YFLM01.0000.00I-1".EPL_FB_OUT_24_I2008_S19Out;
	Cyclic#1.::FBout[25] AT %QW."8YFLM01.0000.00I-1".EPL_FB_OUT_25_I2008_S1AOut;
	Cyclic#1.::FBout[26] AT %QW."8YFLM01.0000.00I-1".EPL_FB_OUT_26_I2008_S1BOut;
	Cyclic#1.::FBout[27] AT %QW."8YFLM01.0000.00I-1".EPL_FB_OUT_27_I2008_S1COut;
	Cyclic#1.::FBout[28] AT %QW."8YFLM01.0000.00I-1".EPL_FB_OUT_28_I2008_S1DOut;
	Cyclic#1.::FBout[29] AT %QW."8YFLM01.0000.00I-1".EPL_FB_OUT_29_I2008_S1EOut;
	Cyclic#1.::FBout[3] AT %QW."8YFLM01.0000.00I-1".EPL_FB_OUT_3_I2008_S04Out;
	Cyclic#1.::FBout[30] AT %QW."8YFLM01.0000.00I-1".EPL_FB_OUT_30_I2008_S1FOut;
	Cyclic#1.::FBout[31] AT %QW."8YFLM01.0000.00I-1".EPL_FB_OUT_31_I2008_S20Out;
	Cyclic#1.::FBout[32] AT %QW."8YFLM01.0000.00I-1".EPL_FB_OUT_32_I2008_S21Out;
	Cyclic#1.::FBout[33] AT %QW."8YFLM01.0000.00I-1".EPL_FB_OUT_33_I2008_S22Out;
	Cyclic#1.::FBout[34] AT %QW."8YFLM01.0000.00I-1".EPL_FB_OUT_34_I2008_S23Out;
	Cyclic#1.::FBout[35] AT %QW."8YFLM01.0000.00I-1".EPL_FB_OUT_35_I2008_S24Out;
	Cyclic#1.::FBout[36] AT %QW."8YFLM01.0000.00I-1".EPL_FB_OUT_36_I2008_S25Out;
	Cyclic#1.::FBout[37] AT %QW."8YFLM01.0000.00I-1".EPL_FB_OUT_37_I2008_S26Out;
	Cyclic#1.::FBout[38] AT %QW."8YFLM01.0000.00I-1".EPL_FB_OUT_38_I2008_S27Out;
	Cyclic#1.::FBout[39] AT %QW."8YFLM01.0000.00I-1".EPL_FB_OUT_39_I2008_S28Out;
	Cyclic#1.::FBout[4] AT %QW."8YFLM01.0000.00I-1".EPL_FB_OUT_4_I2008_S05Out;
	Cyclic#1.::FBout[40] AT %QW."8YFLM01.0000.00I-1".EPL_FB_OUT_40_I2008_S29Out;
	Cyclic#1.::FBout[41] AT %QW."8YFLM01.0000.00I-1".EPL_FB_OUT_41_I2008_S2AOut;
	Cyclic#1.::FBout[42] AT %QW."8YFLM01.0000.00I-1".EPL_FB_OUT_42_I2008_S2BOut;
	Cyclic#1.::FBout[43] AT %QW."8YFLM01.0000.00I-1".EPL_FB_OUT_43_I2008_S2COut;
	Cyclic#1.::FBout[44] AT %QW."8YFLM01.0000.00I-1".EPL_FB_OUT_44_I2008_S2DOut;
	Cyclic#1.::FBout[45] AT %QW."8YFLM01.0000.00I-1".EPL_FB_OUT_45_I2008_S2EOut;
	Cyclic#1.::FBout[46] AT %QW."8YFLM01.0000.00I-1".EPL_FB_OUT_46_I2008_S2FOut;
	Cyclic#1.::FBout[47] AT %QW."8YFLM01.0000.00I-1".EPL_FB_OUT_47_I2008_S30Out;
	Cyclic#1.::FBout[48] AT %QW."8YFLM01.0000.00I-1".EPL_FB_OUT_48_I2008_S31Out;
	Cyclic#1.::FBout[49] AT %QW."8YFLM01.0000.00I-1".EPL_FB_OUT_49_I2008_S32Out;
	Cyclic#1.::FBout[5] AT %QW."8YFLM01.0000.00I-1".EPL_FB_OUT_5_I2008_S06Out;
	Cyclic#1.::FBout[50] AT %QW."8YFLM01.0000.00I-1".EPL_FB_OUT_50_I2008_S33Out;
	Cyclic#1.::FBout[51] AT %QW."8YFLM01.0000.00I-1".EPL_FB_OUT_51_I2008_S34Out;
	Cyclic#1.::FBout[52] AT %QW."8YFLM01.0000.00I-1".EPL_FB_OUT_52_I2008_S35Out;
	Cyclic#1.::FBout[53] AT %QW."8YFLM01.0000.00I-1".EPL_FB_OUT_53_I2008_S36Out;
	Cyclic#1.::FBout[54] AT %QW."8YFLM01.0000.00I-1".EPL_FB_OUT_54_I2008_S37Out;
	Cyclic#1.::FBout[55] AT %QW."8YFLM01.0000.00I-1".EPL_FB_OUT_55_I2008_S38Out;
	Cyclic#1.::FBout[56] AT %QW."8YFLM01.0000.00I-1".EPL_FB_OUT_56_I2008_S39Out;
	Cyclic#1.::FBout[57] AT %QW."8YFLM01.0000.00I-1".EPL_FB_OUT_57_I2008_S3AOut;
	Cyclic#1.::FBout[58] AT %QW."8YFLM01.0000.00I-1".EPL_FB_OUT_58_I2008_S3BOut;
	Cyclic#1.::FBout[59] AT %QW."8YFLM01.0000.00I-1".EPL_FB_OUT_59_I2008_S3COut;
	Cyclic#1.::FBout[6] AT %QW."8YFLM01.0000.00I-1".EPL_FB_OUT_6_I2008_S07Out;
	Cyclic#1.::FBout[60] AT %QW."8YFLM01.0000.00I-1".EPL_FB_OUT_60_I2008_S3DOut;
	Cyclic#1.::FBout[61] AT %QW."8YFLM01.0000.00I-1".EPL_FB_OUT_61_I2008_S3EOut;
	Cyclic#1.::FBout[62] AT %QW."8YFLM01.0000.00I-1".EPL_FB_OUT_62_I2008_S3FOut;
	Cyclic#1.::FBout[63] AT %QW."8YFLM01.0000.00I-1".EPL_FB_OUT_63_I2008_S40Out;
	Cyclic#1.::FBout[64] AT %QW."8YFLM01.0000.00I-1".EPL_FB_OUT_64_I2008_S41Out;
	Cyclic#1.::FBout[65] AT %QW."8YFLM01.0000.00I-1".EPL_FB_OUT_65_I2008_S42Out;
	Cyclic#1.::FBout[66] AT %QW."8YFLM01.0000.00I-1".EPL_FB_OUT_66_I2008_S43Out;
	Cyclic#1.::FBout[67] AT %QW."8YFLM01.0000.00I-1".EPL_FB_OUT_67_I2008_S44Out;
	Cyclic#1.::FBout[68] AT %QW."8YFLM01.0000.00I-1".EPL_FB_OUT_68_I2008_S45Out;
	Cyclic#1.::FBout[69] AT %QW."8YFLM01.0000.00I-1".EPL_FB_OUT_69_I2008_S46Out;
	Cyclic#1.::FBout[7] AT %QW."8YFLM01.0000.00I-1".EPL_FB_OUT_7_I2008_S08Out;
	Cyclic#1.::FBout[70] AT %QW."8YFLM01.0000.00I-1".EPL_FB_OUT_70_I2008_S47Out;
	Cyclic#1.::FBout[71] AT %QW."8YFLM01.0000.00I-1".EPL_FB_OUT_71_I2008_S48Out;
	Cyclic#1.::FBout[72] AT %QW."8YFLM01.0000.00I-1".EPL_FB_OUT_72_I2008_S49Out;
	Cyclic#1.::FBout[73] AT %QW."8YFLM01.0000.00I-1".EPL_FB_OUT_73_I2008_S4AOut;
	Cyclic#1.::FBout[74] AT %QW."8YFLM01.0000.00I-1".EPL_FB_OUT_74_I2008_S4BOut;
	Cyclic#1.::FBout[75] AT %QW."8YFLM01.0000.00I-1".EPL_FB_OUT_75_I2008_S4COut;
	Cyclic#1.::FBout[76] AT %QW."8YFLM01.0000.00I-1".EPL_FB_OUT_76_I2008_S4DOut;
	Cyclic#1.::FBout[77] AT %QW."8YFLM01.0000.00I-1".EPL_FB_OUT_77_I2008_S4EOut;
	Cyclic#1.::FBout[78] AT %QW."8YFLM01.0000.00I-1".EPL_FB_OUT_78_I2008_S4FOut;
	Cyclic#1.::FBout[79] AT %QW."8YFLM01.0000.00I-1".EPL_FB_OUT_79_I2008_S50Out;
	Cyclic#1.::FBout[8] AT %QW."8YFLM01.0000.00I-1".EPL_FB_OUT_8_I2008_S09Out;
	Cyclic#1.::FBout[80] AT %QW."8YFLM01.0000.00I-1".EPL_FB_OUT_80_I2008_S51Out;
	Cyclic#1.::FBout[81] AT %QW."8YFLM01.0000.00I-1".EPL_FB_OUT_81_I2008_S52Out;
	Cyclic#1.::FBout[82] AT %QW."8YFLM01.0000.00I-1".EPL_FB_OUT_82_I2008_S53Out;
	Cyclic#1.::FBout[83] AT %QW."8YFLM01.0000.00I-1".EPL_FB_OUT_83_I2008_S54Out;
	Cyclic#1.::FBout[84] AT %QW."8YFLM01.0000.00I-1".EPL_FB_OUT_84_I2008_S55Out;
	Cyclic#1.::FBout[85] AT %QW."8YFLM01.0000.00I-1".EPL_FB_OUT_85_I2008_S56Out;
	Cyclic#1.::FBout[86] AT %QW."8YFLM01.0000.00I-1".EPL_FB_OUT_86_I2008_S57Out;
	Cyclic#1.::FBout[87] AT %QW."8YFLM01.0000.00I-1".EPL_FB_OUT_87_I2008_S58Out;
	Cyclic#1.::FBout[88] AT %QW."8YFLM01.0000.00I-1".EPL_FB_OUT_88_I2008_S59Out;
	Cyclic#1.::FBout[89] AT %QW."8YFLM01.0000.00I-1".EPL_FB_OUT_89_I2008_S5AOut;
	Cyclic#1.::FBout[9] AT %QW."8YFLM01.0000.00I-1".EPL_FB_OUT_9_I2008_S0AOut;
	Cyclic#1.::FBout[90] AT %QW."8YFLM01.0000.00I-1".EPL_FB_OUT_90_I2008_S5BOut;
	Cyclic#1.::FBout[91] AT %QW."8YFLM01.0000.00I-1".EPL_FB_OUT_91_I2008_S5COut;
	Cyclic#1.::FBout[92] AT %QW."8YFLM01.0000.00I-1".EPL_FB_OUT_92_I2008_S5DOut;
	Cyclic#1.::FBout[93] AT %QW."8YFLM01.0000.00I-1".EPL_FB_OUT_93_I2008_S5EOut;
	Cyclic#1.::FBout[94] AT %QW."8YFLM01.0000.00I-1".EPL_FB_OUT_94_I2008_S5FOut;
	Cyclic#1.::FBout[95] AT %QW."8YFLM01.0000.00I-1".EPL_FB_OUT_95_I2008_S60Out;
	Cyclic#1.::FBout[96] AT %QW."8YFLM01.0000.00I-1".EPL_FB_OUT_96_I2008_S61Out;
	Cyclic#1.::FBout[97] AT %QW."8YFLM01.0000.00I-1".EPL_FB_OUT_97_I2008_S62Out;
	Cyclic#1.::FBout[98] AT %QW."8YFLM01.0000.00I-1".EPL_FB_OUT_98_I2008_S63Out;
	Cyclic#1.::FBout[99] AT %QW."8YFLM01.0000.00I-1".EPL_FB_OUT_99_I2008_S64Out;
END_VAR
```

## Logical view

Binary libraries used (declarations not repeated): operator, runtime, astime, AsIecCon, standard, McAcp6D, AsMath, AsXml, AsBrStr, AsIODiag, LoggingLib, asstring, ArEventLog, AsTCP, FileIO, snprintf, brsystem, AsZip, MTTypes, sys_lib, AsBrMath, McBase, McAcpAx, McPathGen, McAcpTrak, McAxGroup, McAxis, McProgInt, MpAxis, MpBase, MpAudit, MpRecipe, MpFile, MTFilter 5.14.1, MTBasics 5.14.1, CoTrace, MpServer, MpAlarmX, RandLib, SceneView, McPureVAx 5.14.2, SlFreeBase 2.01.0, MTProfile 5.14.1

### Package Logical/Libraries - Global libraries

### Library Logical/Libraries/Prof6DBdlr (IEC)

#### Types.typ - Exported data types
```iecst
TYPE
	ProfBuilderMovePosParTyp : 	STRUCT
		XPos : REAL;
		YPos : REAL;
		ZPos : REAL;
		RxPos : REAL;
		RyPos : REAL;
		RzPos : REAL;
	END_STRUCT;
	ProfBuilderMoveDynParTyp : 	STRUCT
		Vel : REAL;
		Accel : REAL;
		EndVel : REAL;
	END_STRUCT;
	ProfBuilderPlaneParTyp : 	STRUCT
		Path : McAcp6DInPlaneMovePathEnum;
		Mode : McAcp6DMoveModeEnum;
	END_STRUCT;
	ProfBuilderArcParTyp : 	STRUCT
		Angle : REAL;
		Mode : McAcp6DMoveModeEnum;
		Direction : McAcp6DArcDirectionEnum;
	END_STRUCT;
	ProfBuilderMoveTyp :
		(
		profMoveNone,
		profMovePlane,
		profMoveArc,
		profLand
		);
	ProfBuilderMoveParTyp : 	STRUCT
		Positions : ProfBuilderMovePosParTyp;
		Dynamics : ProfBuilderMoveDynParTyp;
		InPlanePar : ProfBuilderPlaneParTyp;
		ArcPar : ProfBuilderArcParTyp;
		MoveType : ProfBuilderMoveTyp;
		WaitTime : UDINT;
		LandPar : McAcp6DLevitationLevelEnum;
	END_STRUCT;
	ProfBuilderParTyp : 	STRUCT
		NumMoves : USINT;
		Moves : ARRAY[0..MAX_NUM_MOVES_ARRAY]OF ProfBuilderMoveParTyp;
	END_STRUCT;
END_TYPE
```

#### Constants.var - Exported constants
```iecst
VAR CONSTANT
	MAX_NUM_MOVES : USINT := 10;
	MAX_NUM_MOVES_ARRAY : USINT := MAX_NUM_MOVES-1;
END_VAR
```

#### Prof6DBdlr.fun - Exported functions and function blocks
```iecst
{REDUND_ERROR} FUNCTION_BLOCK ProfBuilderFb (*TODO: Add your comment here*) (*$GROUP=User,$CAT=User,$GROUPICON=User.png,$CATICON=User.png*)
	VAR_INPUT
		Controller : REFERENCE TO McAcp6DControllerType;
		Reset : BOOL;
		Execute : {REDUND_UNREPLICABLE} BOOL;
		ShId : {REDUND_UNREPLICABLE} USINT;
		Pars : REFERENCE TO ProfBuilderParTyp;
	END_VAR
	VAR_OUTPUT
		Error : {REDUND_UNREPLICABLE} BOOL;
		ErrorID : {REDUND_UNREPLICABLE} DINT;
		Active : {REDUND_UNREPLICABLE} BOOL;
		Moving : {REDUND_UNREPLICABLE} BOOL;
		Done : {REDUND_UNREPLICABLE} BOOL;
	END_VAR
	VAR
		int : {REDUND_UNREPLICABLE} ProfBuilderIntTyp;
	END_VAR
END_FUNCTION_BLOCK
```

#### ProfBuilderFb.st
```iecst
(* TODO: Add your comment here *)
FUNCTION_BLOCK ProfBuilderFb
	CASE int.State OF
		PB_IDLE: 	//******************************************************************************** Idle State
			IF Execute THEN
				Active := TRUE;
				IF Pars.NumMoves > MAX_NUM_MOVES THEN
					Error := TRUE;
					int.State := PB_ERROR;
				ELSE
					int.State := PB_CHECK_IDX;
				END_IF
			END_IF

		PB_CHECK_IDX: 	//******************************************************************************** Checking the Index State

			CASE Pars.Moves[int.idx].MoveType OF
				profMoveNone:
				profMovePlane:
					int.Fbs.InPlaneFb.Controller := ADR(Controller);
					int.Fbs.InPlaneFb.ShuttleID := ShId;
					int.Fbs.InPlaneFb.PositionX := Pars.Moves[int.idx].Positions.XPos;
					int.Fbs.InPlaneFb.PositionY := Pars.Moves[int.idx].Positions.YPos;
					int.Fbs.InPlaneFb.Velocity := Pars.Moves[int.idx].Dynamics.Vel;
					int.Fbs.InPlaneFb.Acceleration := Pars.Moves[int.idx].Dynamics.Accel;
					int.Fbs.InPlaneFb.EndVelocity := Pars.Moves[int.idx].Dynamics.EndVel;
					int.Fbs.InPlaneFb.Mode := Pars.Moves[int.idx].InPlanePar.Mode;
					int.Fbs.InPlaneFb.Path := Pars.Moves[int.idx].InPlanePar.Path;
					int.Fbs.InPlaneFb.Execute := TRUE;
				profMoveArc:
					int.Fbs.ArcFb.Controller := ADR(Controller);
					int.Fbs.ArcFb.ShuttleID := ShId;
					int.Fbs.ArcFb.CenterX := Pars.Moves[int.idx].Positions.XPos;
					int.Fbs.ArcFb.CenterY := Pars.Moves[int.idx].Positions.YPos;
					int.Fbs.ArcFb.Velocity := Pars.Moves[int.idx].Dynamics.Vel;
					int.Fbs.ArcFb.Acceleration := Pars.Moves[int.idx].Dynamics.Accel;
					int.Fbs.ArcFb.EndVelocity := Pars.Moves[int.idx].Dynamics.EndVel;
					int.Fbs.ArcFb.Mode := Pars.Moves[int.idx].ArcPar.Mode;
					int.Fbs.ArcFb.Direction := Pars.Moves[int.idx].ArcPar.Direction;
					int.Fbs.ArcFb.Angle := Pars.Moves[int.idx].ArcPar.Angle;
					int.Fbs.ArcFb.Execute := TRUE;
				profLand:
					int.Fbs.LevitateCtrlFb.Controller := ADR(Controller);
					int.Fbs.LevitateCtrlFb.ShuttleID := ShId;
					int.Fbs.LevitateCtrlFb.Level := Pars.Moves[int.idx].LandPar;
					int.Fbs.LevitateCtrlFb.Execute := TRUE;

			END_CASE;

			IF int.idx = Pars.NumMoves - 1 THEN
				int.State := PB_WAIT_LAST;
			ELSE
				int.State := PB_CMD_MOVE;
			END_IF
		PB_CMD_MOVE: 	//******************************************************************************** Command Move State
			IF int.Fbs.ArcFb.Error OR int.Fbs.InPlaneFb.Error OR int.Fbs.LevitateCtrlFb.Error THEN
				int.ErrorState := int.State;
				int.State := PB_ERROR;
				Error := TRUE;
			ELSE
				CASE Pars.Moves[int.idx].MoveType OF
					profMovePlane:
						IF int.Fbs.InPlaneFb.Acknowledge THEN
							int.Fbs.InPlaneFb.Execute := FALSE;
							int.idx := int.idx + 1;
							int.State := PB_CHECK_IDX;
						END_IF
					profMoveArc:
						IF int.Fbs.ArcFb.Acknowledge THEN
							int.Fbs.ArcFb.Execute := FALSE;
							int.idx := int.idx + 1;
							int.State := PB_CHECK_IDX;
						END_IF
					profLand:
						IF int.Fbs.LevitateCtrlFb.Acknowledge THEN
							int.Fbs.LevitateCtrlFb.Execute := FALSE;
							int.idx := int.idx + 1;
							int.State := PB_CHECK_IDX;
						END_IF
				END_CASE
			END_IF
		PB_WAIT_LAST: 	//******************************************************************************** Waiting for Last Move State
			IF int.Fbs.ArcFb.Error OR int.Fbs.InPlaneFb.Error THEN
				int.ErrorState := int.State;
				int.State := PB_ERROR;
				Error := TRUE;
			ELSE
				CASE Pars.Moves[int.idx].MoveType OF
					profMovePlane:
						IF int.Fbs.InPlaneFb.Done THEN
							int.Fbs.InPlaneFb.Execute := FALSE;
							int.State := PB_DONE;
						END_IF
					profMoveArc:
						IF int.Fbs.ArcFb.Done THEN
							int.Fbs.ArcFb.Execute := FALSE;
							int.State := PB_DONE;
						END_IF
					profLand:
						IF int.Fbs.LevitateCtrlFb.Done THEN
							int.Fbs.LevitateCtrlFb.Execute := FALSE;
							int.State := PB_DONE;
						END_IF
				END_CASE
			END_IF
		PB_DONE: 	//******************************************************************************** Done State
			IF NOT Execute THEN
				int.State := PB_RESET;
			END_IF
		PB_ERROR: 	//******************************************************************************** Error State
			IF Reset THEN
				Reset := FALSE;
				int.State := PB_RESET;
			END_IF
		PB_RESET: 	//******************************************************************************** Reset State
			int.Fbs.ArcFb.Execute := FALSE;
			int.Fbs.InPlaneFb.Execute := FALSE;
			int.Fbs.WaitFb.Execute := FALSE;
			int.Fbs.LevitateCtrlFb.Execute := FALSE;

			int.idx := 0;
			Error := FALSE;
			ErrorID := 0;
			Active := FALSE;
			Done := FALSE;

			IF NOT int.Fbs.ArcFb.Error AND NOT int.Fbs.InPlaneFb.Error AND NOT int.Fbs.LevitateCtrlFb.Error AND NOT int.Fbs.WaitFb.Error THEN
				int.State := PB_IDLE;
			END_IF
	END_CASE

	int.Fbs.ArcFb();
	int.Fbs.InPlaneFb();
	int.Fbs.WaitFb();
	int.Fbs.LevitateCtrlFb();
END_FUNCTION_BLOCK
```

#### ProfBuilderTypes.typ
```iecst
TYPE
	ProfBuilderIntTyp : 	STRUCT
		State : ProfBuilderStatesEnum;
		ErrorState : ProfBuilderStatesEnum;
		idx : USINT;
		Fbs : ProfBuilderFbIntTyp;
	END_STRUCT;
	ProfBuilderFbIntTyp : 	STRUCT
		InPlaneFb : MC_BR_MoveInPlane_Acp6D;
		ArcFb : MC_BR_MoveArcAngle_Acp6D;
		WaitFb : MC_BR_WaitUntilTime_Acp6D;
		LevitateCtrlFb : MC_BR_LevitationCtrl_Acp6D;
	END_STRUCT;
	ProfBuilderStatesEnum :
		(
		PB_IDLE,
		PB_CHECK_IDX,
		PB_CMD_MOVE,
		PB_WAIT_LAST,
		PB_DONE,
		PB_ERROR,
		PB_RESET
		);
END_TYPE
```

### GlobalVars.var
```iecst
(*Constants*)
VAR CONSTANT
	MAX_SHUTTLE_COUNT : USINT := 8; (*Maximum count of shuttles allowed in the system*)
	MAX_SHUTTLE_COUNT_ARRAY : USINT := MAX_SHUTTLE_COUNT-1; (*Maximum count of shuttles - 1 (used for array declaration)*)
	STATION_IS_EMPTY : USINT := 255; (*Index that denotes that a station is empty and available*)
	NUM_PROCESS_STATIONS : USINT := 2;
	NUM_PROCESS_STATION_ARRAY : USINT := NUM_PROCESS_STATIONS-1;
	STATION_1 : USINT := 0;
	STATION_2 : USINT := 1;
END_VAR
(*Global Interfaces*)
VAR
	gShuttleIf : ARRAY[0..MAX_SHUTTLE_COUNT_ARRAY] OF ShuttleIfTyp; (*Interface(s) to control shuttles in the system*)
	gAcp6DCtrlIf : Acp6DCtrlType; (*Interface to control the 6D system as a whole*)
	gMainIf : MainIfTyp := (Cfg:=(ShuttleCount:=1)); (*Main interface to control the system*)
	g6DRecoveryIf : Acp6DRecoveryIfTyp; (*Interface to control the recover process*)
	gProcessInfoIf : ProcessInfoIfTyp; (*Interface to display process related information*)
	gSceneViewerIf : SceneViewerTyp;
	gProcessRecipe : ProcessRecipeTyp;
	gCyclicChlCfgIf : CycChnlCfgIfTyp; (*Interface for the configuration of the cyclic channels*)
	gDanceDemoIf : DanceDemoIfTyp;
	gVariousDemoIf : VariousDemoIf;
	gAntiSloshIf : StationIfTyp;
END_VAR
```

### GlobalTypes.typ
```iecst
(*Main System Interface Types*)

TYPE
	MainIfTyp : 	STRUCT
		Cmd : MainIfCmdTyp;
		Par : MainIfParTyp;
		Cfg : MainIfCfgTyp;
		Sts : MainIfStatusTyp;
	END_STRUCT;
	MainIfCmdTyp : 	STRUCT
		Power : BOOL;
		StartDemoCycle : BOOL;
		StartDefinedDemo : BOOL;
		Stop : BOOL;
		Reset : BOOL;
		StopAllShuttles : BOOL;
	END_STRUCT;
	MainIfParTyp : 	STRUCT
		AutoRecover6D : BOOL;
		DefinedDemo : USINT;
		ProcessDemoTime : TIME;
		DanceDemoTime : TIME;
	END_STRUCT;
	MainIfCfgTyp : 	STRUCT
		ShuttleCount : USINT;
		EnableRobot : BOOL; (*Signals that the Robot should be powered on and used for the control*)
		Enable6D : BOOL; (*Signals that the 6D should be powered on and used for the control*)
	END_STRUCT;
	MainIfStatusTyp : 	STRUCT
		Power6D : BOOL;
		PowerRobot : BOOL;
		Running : BOOL;
		Error : BOOL;
	END_STRUCT;
END_TYPE

(*Process Info Interface*)

TYPE
	ProcessInfoIfTyp : 	STRUCT
		Cmd : ProcessInfoIfCmdTyp;
		Par : ProcessInfoIfParTyp;
		Sts : ProcessInfoIfStsTyp;
	END_STRUCT;
	ProcessInfoIfCmdTyp : 	STRUCT
		Enable : BOOL;
		ResetData : BOOL;
	END_STRUCT;
	ProcessInfoIfParTyp : 	STRUCT
		CurrentProductCount : UDINT;
	END_STRUCT;
	ProcessInfoIfStsTyp : 	STRUCT
		Enabled : BOOL;
		CurrentPPM : REAL;
		CurrentPPH : REAL;
		CurrentBlistersPerMinute : REAL;
		CurrentLayersPerMinute : REAL;
	END_STRUCT;
END_TYPE

(*6D Controller Interface Types*)

TYPE
	Acp6DCmdType : 	STRUCT
		Power : BOOL;
		ErrorReset : BOOL;
		GetErrorInfo : BOOL;
	END_STRUCT;
	Acp6DCtrlType : 	STRUCT
		Cmd : Acp6DCmdType;
		Sts : Acp6DStatusType;
		Par : Acp6DParType;
	END_STRUCT;
	Acp6DParType : 	STRUCT
		Mode : McAcp6DMoveModeEnum;
		PathType : McAcp6DInPlaneMovePathEnum;
		Acceleration : REAL;
		EndVelocity : REAL;
		Velocity : REAL;
		ShuttleID : USINT;
		SegmentID : USINT;
		PositionX : REAL;
		PositionY : REAL;
		MacroEnabled : BOOL;
	END_STRUCT;
	Acp6DStatusType : 	STRUCT
		Error : BOOL;
		ErrorID : DINT;
		Ready : BOOL;
		PowerOn : BOOL;
		ReadyToPowerOn : BOOL;
		ErrorCodes : ARRAY[0..8]OF DINT;
	END_STRUCT;
	Acp6DShuttleInfoType : 	STRUCT
		State : Acp6DShuttleStateInfoTyp;
		Force : Acp6DShuttleForceInfoTyp;
		Position : Acp6DShuttlePosInfoTyp;
	END_STRUCT;
	Acp6DShuttleStateInfoTyp : 	STRUCT
		Valid : BOOL;
		Value : McAcp6DShuttleStateEnum;
	END_STRUCT;
	Acp6DShuttlePosInfoTyp : 	STRUCT
		Valid : BOOL;
		Value : McAcp6DShPositionInfoType;
	END_STRUCT;
	Acp6DShuttleForceInfoTyp : 	STRUCT
		Valid : BOOL;
		Value : McAcp6DShForceInfoType;
	END_STRUCT;
END_TYPE

(*Shuttle Interface Types*)

TYPE
	ShuttleIfCmdTyp : 	STRUCT  (*Commands for controlling a shuttle*)
		Enable : BOOL; (*Command for enabling the control of a shuttle in the process*)
		NextStep : BOOL; (*Command for a shuttle to start the next step in the process*)
		ResetProductInfo : BOOL; (*Command to reset all the product info on a shuttle*)
		Stop : BOOL; (*Command to stop the process for a shuttle*)
		RunProcessDemo : BOOL; (*Command to start the process demo*)
		Reset : BOOL;
	END_STRUCT;
	ShuttleIfCfgMacrosTyp : 	STRUCT  (*Structure of the macro IDs used for operation*)
		RobotProcessMacro : ShuttleIfMacroEnum; (*Macro ID used for sending a shuttle from the load station to the print station*)
	END_STRUCT;
	ShuttleIfParTyp : 	STRUCT  (*Parameters for the shuttle's operation*)
		X : REAL;
		Y : REAL;
		Vel : REAL;
		EndVel : REAL;
		Accel : REAL;
	END_STRUCT;
	ShuttleIfConfigTyp : 	STRUCT  (*Configuration values for a shuttle*)
		ShuttleId : USINT; (*ShuttleID of this shuttle*)
	END_STRUCT;
	ShuttleIfMacroEnum :
		( (*Macro IDs that are used to denote which macro means what*)
		MACRO_ROBOT_PROCESS := 128, (*Macro ID used for sending a shuttle from the load station to the print station*)
		MACRO_ROBOT_PROCESS1, (*Macro ID used for sending a shuttle from the load station to the print station*)
		MACRO_RECOVERY_GROUP0 := 135, (*Macro ID used for recovering the group 0 shuttles*)
		MACRO_RECOVERY_GROUP1 (*Macro ID used for recovering the group 0 shuttles*)
		);
	ShuttleIfDestEnum :
		( (*Destinations for a shuttle to move to*)
		DEST_LOAD,
		DEST_PROCESS_1,
		DEST_PROCESS_2,
		DEST_INSPECT,
		DEST_UNLOAD (*Destination unload*)
		);
	ShuttleProductStateEnum :
		(
		PROD_EMPTY,
		PROD_DOSING,
		PROD_CUBE
		);
	ShuttleIfStatusTyp : 	STRUCT  (*Status information for the shuttle*)
		CurrentDestination : ShuttleIfDestEnum; (*Destination the shuttle is currently moving towards*)
		ShuttleInfo : Acp6DShuttleInfoType; (*CurrentStatus Information about the shuttle*)
		Error : BOOL; (*Shuttle is currently in an error state*)
		ErrorState : ShStateEnum; (*State the shuttle errored at*)
		Recovered : BOOL; (*Shuttle has been recovered*)
		ProductState : ShuttleProductStateEnum;
		LoopCounter : DINT;
		Active : BOOL;
		ProdFill : ARRAY[0..8]OF USINT;
	END_STRUCT;
	ShStateEnum :
		(
		SH_OFF, (*Shuttle is in the off/idle state*)
		SH_INIT, (*Shuttle is in the initilization state*)
		SH_STARTUP, (*Shuttle is in the startup state*)
		SH_IDLE, (*Shuttle is in the idle state after having been recovered*)
		SH_GO_TO_LOAD,
		SH_LOADING,
		SH_CHECK_RECIPE,
		SH_GO_TO_ST_1,
		SH_PREFORM_ST_1,
		SH_GO_TO_ST_2,
		SH_PREFORM_ST_2,
		SH_GO_TO_INSPECT,
		SH_INSPECT,
		SH_GO_TO_UNLOAD,
		SH_UNLOAD,
		SH_STOPPING,
		SH_RESET,
		SH_ERROR := 65535 (*Shuttle is in the error state*)
		);
	ShuttleIfTyp : 	STRUCT  (*Interface for controlling a shuttle*)
		Cmd : ShuttleIfCmdTyp; (*Commands to issue to a shuttle*)
		Par : ShuttleIfParTyp; (*Parameters for the process for this shuttle*)
		Cfg : ShuttleIfConfigTyp; (*Configuration values for this shuttle*)
		Sts : ShuttleIfStatusTyp; (*Status information related to this shuttle*)
	END_STRUCT;
	SceneViewerTyp : 	STRUCT
		Cmds : SceneViewerCmdsTyp;
		Pars : SceneViewerParsTyp;
	END_STRUCT;
	SceneViewerCmdsTyp : 	STRUCT
		Record : BOOL;
		Clear : BOOL;
	END_STRUCT;
	SceneViewerParsTyp : 	STRUCT
		LineColor : SceneViewerColorTyp;
	END_STRUCT;
	SceneViewerColorTyp : 	STRUCT
		Red : REAL;
		Green : REAL;
		Blue : REAL;
	END_STRUCT;
END_TYPE

(*Recovery Interface Type*)

TYPE
	Acp6DRecoveryIfTyp : 	STRUCT
		Cmd : Acp6DRecoveryCmdTyp;
		Par : Acp6DRecoveryParTyp;
		Sts : Acp6DRecoveryStsTyp;
	END_STRUCT;
	Acp6DRecoveryCmdTyp : 	STRUCT
		Recover : BOOL;
		Reset : BOOL;
	END_STRUCT;
	Acp6DRecoveryParTyp : 	STRUCT
		AutoDrivePositions : ARRAY[0..MAX_SHUTTLE_COUNT_ARRAY]OF Acp6DAutoDrivePosTyp;
		Vel : REAL;
		Accel : REAL;
	END_STRUCT;
	Acp6DRecoveryStsTyp : 	STRUCT
		Recovering : BOOL;
		ReadyToStartProc : BOOL;
		Done : BOOL;
		ShuttlesRecovered : BOOL;
		Error : BOOL;
	END_STRUCT;
	Acp6DAutoDrivePosTyp : 	STRUCT
		ShIdx : USINT;
		X : REAL;
		Y : REAL;
	END_STRUCT;
END_TYPE

(*Process Demo Recipe Types*)

TYPE
	ProcessRecipeTyp : 	STRUCT
		General : ProcessRecipeGenTyp;
		Load : ProcessRecipeLoadTyp;
		Unload : ProcessRecipeLoadTyp;
		St1 : ProcessRecipeStationTyp;
		St2 : ProcessRecipeStationTyp;
		Inspect : ProcessRecipeStationTyp;
	END_STRUCT;
	ProcessRecipeGenTyp : 	STRUCT
		St1St2Cycles : USINT;
		Velocity : REAL;
		Accel : REAL;
		Decel : REAL;
	END_STRUCT;
	ProcessRecipeLoadTyp : 	STRUCT
		StartPos : StationPositionTyp;
		EndPos : StationPositionTyp;
	END_STRUCT;
	ProcessRecipeStationTyp : 	STRUCT
		MacroId : USINT;
		DwellTime : TIME;
		OperationPos : StationPositionTyp;
		ExitPos : StationPositionTyp;
	END_STRUCT;
END_TYPE

(*6D Cyclic Channel Configurationi Types*)

TYPE
	CycChnlCfgIfTyp : 	STRUCT
		Cmds : CycChnlCfgCmdsIfTyp;
		Pars : CycChnlCfgParsIfTyp;
		Sts : CycChnlCfgStsIfTyp;
	END_STRUCT;
	CycChnlCfgCmdsIfTyp : 	STRUCT
		Config : BOOL;
	END_STRUCT;
	CycChnlCfgParsIfTyp : 	STRUCT
		LoadShuttleIdx : USINT;
		UnloadShuttleIdx : USINT;
	END_STRUCT;
	CycChnlCfgStsIfTyp : 	STRUCT
		Ready : BOOL;
		Configuring : BOOL;
		Error : BOOL;
	END_STRUCT;
END_TYPE

(***********************Station Types*)

TYPE
	StationIfTyp : 	STRUCT
		Cmd : StationIfCmdTyp; (*Commands to a station*)
		Par : {REDUND_UNREPLICABLE} StationIfParTyp; (*Parameters for the station's operation*)
		Cfg : StationIfCfgTyp; (*Configuration values for the station*)
		Sts : StationIfStsTyp; (*Status of the station*)
	END_STRUCT;
	StationIfCmdTyp : 	STRUCT
		Enable : BOOL; (*Enables the process station*)
		Process : BOOL; (*Start a process for the station with the defined shuttle index*)
		Reset : BOOL; (*Resets the process from an any state*)
		LocalOverride : BOOL; (*Denotes that local settings can be overwritten from global*)
	END_STRUCT;
	StationIfCfgTyp : 	STRUCT
		StationPos : StationPositionTyp; (*Station's center world position*)
	END_STRUCT;
	StationIfParTyp : 	STRUCT
		ShuttleIdx : USINT; (*Index in the gShuttle array for the shuttle in question*)
	END_STRUCT;
	StationIfStsTyp : 	STRUCT
		Enabled : BOOL; (*Signal denoting the station is enabled and in an operational state*)
		Processing : BOOL; (*Signal denoting the station is currently operating on a shuttle*)
		Done : BOOL; (*Signal denoting the current operation has completed*)
		ReadyForNewShuttle : BOOL; (*Signal denoting the station is ready for a new shuttle*)
		Error : BOOL; (*Signal denoting the station has an error present*)
	END_STRUCT;
	StationPositionTyp : 	STRUCT
		X : REAL; (*Station's Global X position*)
		Y : REAL; (*Station's Global Y position*)
	END_STRUCT;
	FillStationEnum :
		(
		ST_UNDEF,
		ST1,
		ST2,
		ST3,
		ST4
		);
END_TYPE

(*Dance Demo If*)

TYPE
	DanceDemoIfTyp : 	STRUCT
		Cmd : DanceDemoCmdTyp;
		Par : DanceDemoParTyp;
		Sts : DanceDemoStsTyp;
	END_STRUCT;
	DanceDemoCmdTyp : 	STRUCT
		Run : BOOL;
		Reset : BOOL;
	END_STRUCT;
	DanceDemoParTyp : 	STRUCT
		DemoTime : TIME; (*How long each demo should run for*)
	END_STRUCT;
	DanceDemoStsTyp : 	STRUCT
		Running : BOOL;
		Error : BOOL;
	END_STRUCT;
END_TYPE

(**************************** Various Demo Types*)

TYPE
	VariousDemoTypesEnum :
		(
		VAR_DEMO_SLIDE,
		VAR_DEMO_MIX,
		VAR_DEMO_WEIGH,
		VAR_DEMO_WAVE,
		VAR_DEMO_FORCE,
		VAR_DEMO_ANTI_SLOSH,
		VAR_DEMO_LAND,
		VAR_DEMO_CYCLE,
		VAR_DEMO_GENERIC_MOVEMENT
		);
	VariousDemoIf : 	STRUCT
		Cmd : VariousDemoIfCmdTyp;
		Par : VariousDemoIfParTyp;
		Sts : VariousDemoIfStsTyp;
	END_STRUCT;
	VariousDemoIfParTyp : 	STRUCT
		Demo : VariousDemoTypesEnum;
	END_STRUCT;
	VariousDemoIfCmdTyp : 	STRUCT
		RunDemo : BOOL;
		ChangeDemo : BOOL;
		Stop : BOOL;
		Reset : BOOL;
	END_STRUCT;
	VariousDemoIfStsTyp : 	STRUCT
		CurrentDemo : VariousDemoTypesEnum;
		Active : BOOL;
		Error : BOOL;
		Running : BOOL;
	END_STRUCT;
END_TYPE
```

### Package Logical/Source/ShuttleCtrl - Package that contains code for controlling individual shuttles

### Program Logical/Source/ShuttleCtrl/ShCtrl (IEC)

#### Types.typ
```iecst
TYPE
	ShFbsTyp : 	STRUCT
		ShRunMacroFb : MC_BR_MacroRun_Acp6D; (*Execute a macro on the current shuttle*)
		MovePlane : MC_BR_MoveInPlane_Acp6D;
		Stop : MC_BR_Stop_Acp6D;
	END_STRUCT;
END_TYPE
```

#### Variables.var
```iecst
VAR
	i : USINT; (*Loop index*)
	shState : ARRAY[0..MAX_SHUTTLE_COUNT_ARRAY] OF ShStateEnum;
	shFbs : ARRAY[0..MAX_SHUTTLE_COUNT_ARRAY] OF ShFbsTyp;
	pDebugIf : REFERENCE TO ShuttleIfTyp;
	pDebugFbs : REFERENCE TO ShFbsTyp;
	pDebugState : REFERENCE TO ShStateEnum;
	debugIdx : USINT;
	logArgs : ARRAY[0..3] OF UDINT;
END_VAR
```
